    AXIS_COMBINED_VERTICAL_CALIBRATION : UINT := 25;
    AXIS_COMBINED_VERTICAL_SAMPLE : UINT :=26;
    AXIS_COMBINED_VERTICAL_VIRTUAL : UINT :=27;
    
    AXIS_HORIZONTAL_CALIBRATION : UINT :=28;
    AXIS_HORIZONTAL_SAMPLE : UINT :=29;
    AXIS_HORIZONTAL_VIRTUAL : UINT :=30;
    

END_VAR

// ---- tc_mca_std_lib/GVLs/GVL.TcGVL
VAR_GLOBAL
    // Semantic version in machine-readable format.
    // Update it and commit it immediatly before setting a tag
    nVersionMajor: UINT := 2; // Major Version
    nVersionMinor: UINT := 0; // Minor Version
    nVersionPatch: UINT := 2; // Patch level
    astAxes: ARRAY [1..GVL_APP.nAXIS_NUM] OF ST_AxisStruct; //Array of ST_AxisStruct for holding axis parameters and controls
    astPneumaticAxes: ARRAY [1..GVL_APP.nPNEUMATIC_AXIS_NUM] OF ST_PneumaticAxisStruct; //Array of ST_PneumaticAxisStruct for holding pneumatic axis parameters and controls
    iAxis: UINT; //Index for for loops while going through axes
    iPneumaticAxis: UINT := 1; //Index for for loops while going through pneumatic axes
    fbGetCurTaskIndex: GETCURTASKINDEX;
    bLocalMode: BOOL;
END_VAR

VAR_GLOBAL CONSTANT
    nMAX_AXIS_NAME: UINT := 32;
END_VAR

VAR_GLOBAL PERSISTENT
    astAxesPersistent: ARRAY [1..GVL_APP.nAXIS_NUM] OF ST_AxisPersistent;
END_VAR

// ---- POUs/MAIN.TcPOU
PROGRAM MAIN
VAR
    sVersion: STRING := '1.0.0';
    aIAxes: ARRAY [1..GVL_APP.nAXIS_NUM] OF I_Axis;
    afbAxes: ARRAY [1..GVL_APP.nAXIS_NUM] OF FB_Axis;
    afbPneumaticAxes: ARRAY [1..GVL_APP.nPNEUMATIC_AXIS_NUM] OF FB_PneumaticAxis;
    hmiAxisSelection: INT := 1; //Not possible to use local hmi variables for array indexes
    hmiPneumaticAxisSelection: INT := 1;
//Startup, Shutdown and UPS
    fbUPS: FB_S_UPS_CX51x0;
    eUpsMode: E_S_UPS_Mode := eSUPS_WrPersistData_Shutdown;
    eStartUp: (eColdStart, eReadAxisFeedbackType, eCheckReadDone, eExecuteRestore, eCheckRestore, eFinishRestore);
    bPositionRestoreDone: BOOL := FALSE;
    bRestoreExecute: BOOL := FALSE;
    bExecuteReadEncRefSys: BOOL := FALSE;
    nRetry: INT;
    iAxes: UINT; //index for for loops in Position recovery actions
    afbReadEncRefSys: ARRAY [1..GVL_APP.nAXIS_NUM] OF MC_ReadParameter;
    afbSetPosition: ARRAY [1..GVL_APP.nAXIS_NUM] OF MC_SetPosition;
    afbReadPositionBias: ARRAY [1..GVL_APP.nAXIS_NUM] OF MC_ReadParameter;
    afbWritePositionBias: ARRAY [1..GVL_APP.nAXIS_NUM] OF MC_WriteParameter;
    fbGetDeviceIdentification: FB_GetDeviceIdentificationEx;
    
    
    
END_VAR

VAR PERSISTENT
    bRestoreOnStartup: BOOL;
END_VAR

POSITION_RECOVERY();
PROG();
AXES();

ACTION AXES:
//First cycle, assign FB_axis to interface array
IF _TaskInfo[fbGetCurTaskIndex.index].FirstCycle THEN
    FOR GVL.iAxis := 1 TO GVL_APP.nAXIS_NUM DO
        afbAxes[GVL.iAxis].stAxis REF= astAxes[GVL.iAxis];
        aIAxes[GVL.iAxis] := afbAxes[GVL.iAxis];
    END_FOR
    //Custom axis types defined and linked to aiAxes here
      //FB_CustomAxis extends FB_axis
        //fbCustomAxis.stAxis REF= astAxes[x];
        //aIAxes[x] := fbCustomAxis;
END_IF

//Execute FB_Axis logic
FOR GVL.iAxis := 1 TO GVL_APP.nAXIS_NUM DO
    aIAxes[GVL.iAxis].Run();
END_FOR

//Execute Pneumatic Axis logic
FOR GVL.iPneumaticAxis := 1 TO GVL_APP.nPNEUMATIC_AXIS_NUM DO
    afbPneumaticAxes[GVL.iPneumaticAxis](stPneumaticAxisStruct := GVL.astPneumaticAxes[GVL.iPneumaticAxis]);
END_FOR
END_ACTION

ACTION CHECK_UPS:
fbUPS(eUpsMode := eUpsMode);

FOR iAxes := 1 TO GVL_APP.nAXIS_NUM DO
    //Read encoder position BIAS
    IF astAxes[iAxes].stStatus.bAxisInitialized THEN
        afbReadPositionBias[iAxes](Axis := GVL.astAxes[iAxes].Axis,
                        Enable := TRUE,
                        ReadMode:= READMODE_CYCLIC,
                        ParameterNumber := E_AxisParameters.AxisEncoderOffset);
    END_IF
END_FOR

IF eGlobalSUpsState = eSUPS_PowerFailure THEN
    //first cycle of powerfailure
    //execute code that should only be done once with each powerfailure, i.e. increase powerfailure counter
    bRestoreOnStartup := TRUE;
    STORE_PERSISTENT();
    RETURN;
ELSIF eGlobalSUpsState <> eSUPS_PowerOK THEN
    //next cycles of powerfailure
    //skip regular code execution for the remaining cycles of the powerfailure/writing of persistent data/quick shutdown...
    RETURN;
END_IF
END_ACTION

ACTION POSITION_RECOVERY:
fbGetDeviceIdentification(bExecute := TRUE);
IF (fbGetDeviceIdentification.stDevIdent.strHardwareSerialNo <> '') THEN
    CHECK_UPS();
    RESTORE_POSITIONS();
END_IF
END_ACTION

ACTION PROG:
//Get task index for Axes parameters initialization.
GVL.fbGetCurTaskIndex();

//Call the programs that are defined in the "Application Specific" folder.
//Create as many programs in that folder as axes and applications you have or need

//Axes initial parameters and program
//Axis_Template();
//Pneumatics_Template();

//Application program calls
//Application_Template();
PLC_SAFETY_LOGIC();

Horizontal_Translation();
Vertical_Translation_Y2();
Vertical_Translation_Y1();
Rotation();

Combined_Vertical();


Drad_External();
Drad_Internal();
Doff_Angled();
Doff_Parallel();
Dtank_Internal_Offset_Angle();
Dtank_Length();
Dtank_Pivot_To_Window();
Delta();
Tau();
Drad();
Measurement_Angle();
Rotation_Calibration();
Rotation_Sample();
Horizontal_Calibration();
Horizontal_Sample();
Combined_Vertical_Calibration();
Combined_Vertical_Sample();
Measurement_Angle_Offset();


Rotation_Virtual();
Combined_Vertical_Virtual();
Horizontal_Virtual();




INTER_LOGIC();
VirtualSpeedOverrides();
//Slit setup
Slit_North();
Slit_South();
Slit_East();
Slit_West();
Slit_3();

Inclinometer();
END_ACTION

ACTION RESTORE_POSITIONS:
//This ACT will restore the position of an incremental axis on startup with the act position it read before losing power.
//It checks the type of axis, 0=incremental, and that the axis was stationary at shut down.
//Because 0 equates to incremental we also need to check that the data is valid, otherwise by default it would restore all axes.
//By default an axis will not restore the position unless it is set to opt-in, i.e. GVL.aAxes[iAxes].stConfig.eRestorePosition is non-zero.
//This needs to be initialised somewhere in TwinCAT code otherwise it will not be available at start up.
//A restore will only be performed on a loss of power, this code shouldn't make any changes on a reset cold, a rest origin or a download.
//There is a enum to allow for different types of restore modes, currently only one is implemented.
//0 'DontRestore'
//1 'RestoreWithoutHome' -restores the position using a set position fb and does not set the home bit in the axis struct.
//Note from Beckhoff: "A maximum of 1 MB persistent data can be reliably saved over the entire service life."
//Encoder Reference system types: https://infosys.beckhoff.com/english.php?content=../content/1033/tf50x0_tc3_nc_ptp/3439907723.html&id=
//INCREMENTAL=0;
//ABSOLUTE=1;
//ABSOLUTE (modulo)=2;
//ABSOLUTE MULTITURN RANGE (with single overflow)=3;
//INCREMENTAL (singleturn absolute)=4;
//ABSOLUTE SINGLETURN RANGE (with single overflow)=5;


IF bRestoreOnStartup AND eGlobalSUpsState = eSUPS_PowerOK THEN
    bRestoreOnStartup := FALSE;
    bRestoreExecute := TRUE;
END_IF

//Upon startup bPositionRestoreDone will be set to FALSE, after successfully completing the following code it will be set TRUE
//and should stay TRUE for the rest of the time the PLC is operational, thus this routine should only be completed once.
IF bRestoreExecute AND NOT bPositionRestoreDone THEN
    //Cycle through function blocks that read the encoder reference system i.e. whether axis is incremental or absolute
    FOR iAxes := 1 TO GVL_APP.nAXIS_NUM DO
         afbReadEncRefSys[iAxes](
            Axis := GVL.astAxes[iAxes].Axis,
            ParameterNumber := MC_AxisParameter.AxisEncoderReferenceSystem,
            ReadMode := E_READMODE.READMODE_ONCE);
    END_FOR

    //Cycle through set position and MC_WritePArameter function blocks for each axis
    FOR iAxes := 1 TO GVL_APP.nAXIS_NUM DO
        afbSetPosition[iAxes](
            Axis := GVL.astAxes[iAxes].Axis,
            Position := astAxesPersistent[iAxes].fPositionAtShutdown);

        afbWritePositionBias[iAxes](
            Axis:= GVL.astAxes[iAxes].Axis,
            ParameterNumber:= E_AxisParameters.AxisEncoderOffset,
            Value:= astAxesPersistent[iAxes].fEncoderBiasAtShutdown);
    END_FOR

    CASE eStartUp OF
        eColdStart:
            //First cycle of the PLC, do nothing just give one cycle for variables to initialise
            IF NOT bPositionRestoreDone THEN
                eStartUp := eReadAxisFeedbackType;
                nRetry := 0;
            END_IF

        eReadAxisFeedbackType:
            //Exectute the function blocks to read the encoder reference system (0=inc OR 1=ABS)
            FOR iAxes := 1 TO GVL_APP.nAXIS_NUM DO
                afbReadEncRefSys[iAxes].Enable := TRUE;
                eStartUp := eCheckReadDone;
            END_FOR

        eCheckReadDone:
            //Check the encoder reference system has been read for all axis -> if busy then continue with PLC cycle and check again next time.
            //If afbReadEncRefSys not started then go back a step.
            //If any axes result in an error the code will get stuck here, this happens if GVL_APP.nAXIS_NUM is not set correctly
            FOR iAxes := 1 TO GVL_APP.nAXIS_NUM DO
                IF NOT afbReadEncRefSys[iAxes].Valid THEN
                    IF afbReadEncRefSys[iAxes].Busy THEN
                        //Exit MAIN.STARTUP Action and wait till next cycle, needs to cycle through whole program in order for data to update
                        RETURN;
                    ELSE
                        //Sometimes the code gets here and the afbReadEncRefSys[iAxes] misses the rising edge. If  the code gets here it means
                        //valid=FALSE and .busy=FALSE which indicateds the FB probably hasn't started and thus needs to see a rising edge.
                        //Set execute to low, Exit MAIN.STARTUP and go back a step in the CASE statement.
                        afbReadEncRefSys[iAxes].Enable := FALSE;
                        eStartUp := eReadAxisFeedbackType;
                        nRetry := nRetry + 1; //counter used for troubleshooting to see how many cycles it takes before afbReadEncRefSys function blocks are read correctly
                        RETURN;
                    END_IF
                END_IF
            END_FOR
            //If the code gets here all axes have .valid=TRUE for all axes
            eStartUp := eExecuteRestore;

        eExecuteRestore:
            //Execute position and encoder BIAS restore by setting Execute = TRUE
           FOR iAxes := 1 TO GVL_APP.nAXIS_NUM DO
                IF GVL.astAxes[iAxes].stConfig.eRestorePosition = E_RestorePosition.eRestoreWithoutHome THEN
                    //Restore position value for incremental encoders
                    IF NOT astAxesPersistent[iAxes].bMovingAtShutdown AND
                    (afbReadEncRefSys[iAxes].Value = 0 OR
                     afbReadEncRefSys[iAxes].Value = 2 OR
                     afbReadEncRefSys[iAxes].Value = 4) THEN
                       afbSetPosition[iAxes].Execute := TRUE;
                    //Restore encoder position BIAS for absolute encoders
                    ELSIF afbReadEncRefSys[iAxes].Value = 1 OR
                    afbReadEncRefSys[iAxes].Value = 3 OR
                    afbReadEncRefSys[iAxes].Value = 5 THEN
                       afbWritePositionBias[iAxes].Execute := TRUE;
                    END_IF
                ELSE
                    RETURN;
                END_IF
            END_FOR
            eStartUp := eCheckRestore;


        eCheckRestore:
            //Check the set position and write enocder BIAS fbs are finished
            //Nothing actually happens if the restore is not done, the code just returns from here each cycle and the
            //bPositionRestoreDone will never get set to TRUE and will take up cycle time
            FOR iAxes := 1 TO GVL_APP.nAXIS_NUM DO
                IF GVL.astAxes[iAxes].stConfig.eRestorePosition = E_RestorePosition.eRestoreWithoutHome THEN
                    IF NOT astAxesPersistent[iAxes].bMovingAtShutdown AND
                    (afbReadEncRefSys[iAxes].Value = 0 OR
                     afbReadEncRefSys[iAxes].Value = 2 OR
                     afbReadEncRefSys[iAxes].Value = 4) THEN
                        IF NOT afbSetPosition[iAxes].Done THEN
                            afbSetPosition[iAxes].Execute := FALSE;
                            eStartUp := eExecuteRestore;
                            RETURN;
                        END_IF
                     ELSIF afbReadEncRefSys[iAxes].Value = 1 OR
                     afbReadEncRefSys[iAxes].Value = 3 OR
                     afbReadEncRefSys[iAxes].Value = 5 THEN
                        IF NOT afbWritePositionBias[iAxes].Done THEN
                            afbWritePositionBias[iAxes].Execute := FALSE;
                            eStartUp := eExecuteRestore;
                            RETURN;
                        END_IF
                    END_IF
                ELSE
                    RETURN;
                END_IF
            END_FOR
            eStartUp :=  eFinishRestore;

        eFinishRestore:
            //Remove execute = TRUE for afbRestorePosition and fbWritePositionBias
            FOR iAxes := 1 TO GVL_APP.nAXIS_NUM DO
                afbSetPosition[iAxes].Execute := FALSE;
                afbWritePositionBias[iAxes].Execute := FALSE;
                bPositionRestoreDone := TRUE;
                bRestoreExecute := FALSE;
            END_FOR
    END_CASE
END_IF
END_ACTION

ACTION STORE_PERSISTENT:
FOR iAxes := 1 TO GVL_APP.nAXIS_NUM DO
    //Store Position beofre shutdown
    astAxesPersistent[iAxes].fPositionAtShutdown := GVL.astAxes[iAxes].Axis.NcToPlc.ActPos;

    //Store encoder position BIAS at shutdown
    astAxesPersistent[iAxes].fEncoderBiasAtShutdown := afbReadPositionBias[iAxes].Value;

    //Store value of moving at shutdown
    IF GVL.astAxes[iAxes].Axis.Status.StandStill OR GVL.astAxes[iAxes].Axis.Status.Disabled THEN
        astAxesPersistent[iAxes].bMovingAtShutdown := FALSE;
    ELSE
        astAxesPersistent[iAxes].bMovingAtShutdown := TRUE;
    END_IF
END_FOR
END_ACTION

END_PROGRAM

// ---- tc_mca_std_lib/POUs/Motion/FB_Axis.TcPOU
//Function block to run a virtual drive with Nc
FUNCTION_BLOCK FB_Axis IMPLEMENTS I_axis
VAR
    _stAxis: REFERENCE TO ST_AxisStruct; // Local property pointer for axis structure
    astMcStatus: ARRAY[1..nMCSTATUS_ARRAY_SIZE] OF POINTER TO ST_McStatus; //Array of all MC status signals defined in FB_init

    fbPower: MC_Power;
    stMcStatusPower: ST_McStatus;

    fbStop: MC_Stop;
    stMcStatusStop: ST_McStatus;

    fbHalt: MC_Halt;
    stMcStatusHalt: ST_McStatus;

    fbReset: MC_Reset;
    stMcStatusReset: ST_McStatus;

    fbMoveAbsolute: MC_MoveAbsolute;
    stMcStatusMoveAbsolute: ST_McStatus;

    fbMoveRelative: MC_MoveRelative;
    stMcStatusMoveRelative: ST_McStatus;

    fbMoveVelocity: MC_MoveVelocity;
    stMcStatusMoveVelocity: ST_McStatus;

    fbMoveModulo: MC_MoveModulo;
    stMcStatusMoveModulo: ST_McStatus;

    fbHome: FB_Homing;
    stMcStatusHome: ST_McStatus;

    fbReadParameter: MC_ReadParameter;
    stMcStatusReadParameter: ST_McStatus;

    fbWriteParameter: MC_WriteParameter;
    stMcStatusWriteParameter: ST_McStatus;

    fbGearIn: MC_GearIn;
    stMcStatusGearIn: ST_McStatus;

    fbGearOut: MC_GearOut;
    stMcStatusGearOut: ST_McStatus;

    stMasterAxis: ST_GearAxis := (nIndex := 1, fRatio := 0);
    nSlaveAxesIndex: UINT;
    nAxisIndex: UINT;
    nMultiMastersAxesIndex: UINT;

    fbGearInMultiMaster: MC_GearInMultiMaster;
    stMcStatusGearInMultiMaster: ST_McStatus;

    //Variables for holding limits during homing
    bWaitForStopAfterLimitHit: BOOL := FALSE;
    fbRemovePowerTimer: TOF;

    //Dedicated NC parameter read FBs
    fbReadAxisVeloManSlow: MC_ReadParameter;
    fbReadAxisVeloManFast: MC_ReadParameter;
    fbReadHomingVelToCam: MC_ReadParameter;
    fbReadHomingVelFromCam: MC_ReadParameter;
    fbReadAxisVeloMax: MC_ReadParameter;
    fbReadAxisMaxAcc: MC_ReadParameter;
    fbReadAxisMaxDec: MC_ReadParameter;
    fbReadAxisAcc: MC_ReadParameter;
    fbReadAxisDec: MC_ReadParameter;
    fbReadEnMinSoftPosLimit: MC_ReadParameter;
    fbReadEnMaxSoftPosLimit: MC_ReadParameter;
    fbReadMinSoftPosLimit: MC_ReadParameter;
    fbReadMaxSoftPosLimit: MC_ReadParameter;
    fbReadEnPositionLagMonitoring: MC_ReadParameter;
    fbReadAxisMaxPosLagValue: MC_ReadParameter;
    fbReadEnTargetPositionMonitoring: MC_ReadParameter;
    fbReadTargetPositionWindow: MC_ReadParameter;

    //Edge detection triggers for statuses
    fbDoneRTrig: R_TRIG;
    fbErrorRTrig: R_TRIG;
    fbCommandAbortedRTrig: R_TRIG;
    fbInVelocityRTrig: R_TRIG;
    fbInVelocityFTrig: F_TRIG;
    fbExecuteRTrig: R_TRIG;
    fbStopFinishedRiseEdge: R_TRIG;
    fbHaltFinishedRiseEdge: R_TRIG;
    fbResetFinishedRiseEdge: R_TRIG;

END_VAR
VAR CONSTANT
    nRATIO_DENOMINATOR_DEFAULT: UINT := 1;
    nNO_GEARING: UINT := 0;
    nMCSTATUS_ARRAY_SIZE: UINT := 13;
    nMULTI_MASTER_MAX_AXES: UINT := 4;
END_VAR

METHOD EndOfCycle : BOOL

_stAxis.stControl.bExecute := FALSE;
END_METHOD

METHOD FB_init : BOOL
VAR_INPUT
    bInitRetains: BOOL; // if TRUE, the retain variables are initialized (warm start / cold start)
    bInCopyCode: BOOL; // if TRUE, the instance afterwards gets moved into the copy code (online change)
END_VAR

//Copy address locations for statuses to an array to allow for easier checking of statuses
astMcStatus[1] := ADR(stMcStatusPower);
astMcStatus[2] := ADR(stMcStatusStop);
astMcStatus[3] := ADR(stMcStatusHalt);
astMcStatus[4] := ADR(stMcStatusReset);
astMcStatus[5] := ADR(stMcStatusMoveAbsolute);
astMcStatus[6] := ADR(stMcStatusMoveRelative);
astMcStatus[7] := ADR(stMcStatusMoveVelocity);
astMcStatus[8] := ADR(stMcStatusMoveModulo);
astMcStatus[9] := ADR(stMcStatusHome);
astMcStatus[10] := ADR(stMcStatusGearInMultiMaster);
astMcStatus[11] := ADR(stMcStatusGearOut);
astMcStatus[12] := ADR(stMcStatusReadParameter);
astMcStatus[13] := ADR(stMcStatusWriteParameter);
END_METHOD

METHOD mControl_GearInMultiMaster : ST_McStatus

fbGearInMultiMaster.Options.AdvancedSlaveDynamics := TRUE;
fbGearInMultiMaster.Options.SyncMode := E_GearInMultiMasterSyncMode.POSSYNC2;
IF _stAxis.stControl.eCommand = E_MotionFunctions.eGearInMultiMaster THEN
    fbGearInMultiMaster.Enable := _stAxis.stControl.bExecute;
END_IF

IF _stAxis.stControl.eCommand = E_MotionFunctions.eGearInMultiMaster AND _stAxis.stControl.bExecute AND NOT _stAxis.Axis.Status.Coupled THEN
    //Latch master references
    FOR nMultiMastersAxesIndex := 1 TO nMULTI_MASTER_MAX_AXES DO
        IF _stAxis.stConfig.astMultiMasterAxis[nMultiMastersAxesIndex].nIndex > 0 AND _stAxis.stConfig.astMultiMasterAxis[nMultiMastersAxesIndex].nIndex <= GVL_APP.nAXIS_NUM THEN
            _stAxis.stConfig.astMultiMasterAxisLatched[nMultiMastersAxesIndex].nIndex := _stAxis.stConfig.astMultiMasterAxis[nMultiMastersAxesIndex].nIndex;
        END_IF
    END_FOR
    //Latch gear ratios
    FOR nMultiMastersAxesIndex := 1 TO nMULTI_MASTER_MAX_AXES DO
        _stAxis.stConfig.astMultiMasterAxisLatched[nMultiMastersAxesIndex].fRatio := _stAxis.stConfig.astMultiMasterAxis[nMultiMastersAxesIndex].fRatio;
    END_FOR
    //Transfer gear ratios to FB
    fbGearInMultiMaster.GearRatio1 := _stAxis.stConfig.astMultiMasterAxisLatched[1].fRatio;
    fbGearInMultiMaster.GearRatio2 := _stAxis.stConfig.astMultiMasterAxisLatched[2].fRatio;
    fbGearInMultiMaster.GearRatio3 := _stAxis.stConfig.astMultiMasterAxisLatched[3].fRatio;
    fbGearInMultiMaster.GearRatio4 := _stAxis.stConfig.astMultiMasterAxisLatched[4].fRatio;
    fbGearInMultiMaster.Enable := TRUE;
END_IF

fbGearInMultiMaster(Slave := _stAxis.Axis,
    Master1 := GVL.astAxes[_stAxis.stConfig.astMultiMasterAxisLatched[1].nIndex].Axis,
    Master2 := GVL.astAxes[_stAxis.stConfig.astMultiMasterAxisLatched[2].nIndex].Axis,
    Master3 := GVL.astAxes[_stAxis.stConfig.astMultiMasterAxisLatched[3].nIndex].Axis,
    Master4 := GVL.astAxes[_stAxis.stConfig.astMultiMasterAxisLatched[4].nIndex].Axis);
fbGearInMultiMaster.Enable:= FALSE;

IF fbGearInMultiMaster.InGear THEN
    mStatus_MultiGearing();
END_IF

IF fbGearInMultiMaster.Error THEN
    fbGearInMultiMaster.Enable := FALSE;
END_IF

mControl_GearInMultiMaster.Active := fbGearInMultiMaster.Active;
mControl_GearInMultiMaster.Done := fbGearInMultiMaster.InGear;
mControl_GearInMultiMaster.Busy := fbGearInMultiMaster.Busy;
mControl_GearInMultiMaster.Error := fbGearInMultiMaster.Error;
mControl_GearInMultiMaster.ErrorID := fbGearInMultiMaster.ErrorID;
mControl_GearInMultiMaster.CommandAborted := fbGearInMultiMaster.CommandAborted;

IF fbGearInMultiMaster.Error THEN
    _stAxis.stError.nGearInMultiMasterErrorID := fbGearInMultiMaster.ErrorID; //Set the error
END_IF
END_METHOD

METHOD mControl_GearOut : ST_McStatus

IF _stAxis.stControl.eCommand = E_MotionFunctions.eGearOut THEN
    fbGearOut.Execute := _stAxis.stControl.bExecute;
END_IF

fbGearOut(Slave := _stAxis.Axis);
fbGearOut.Execute := FALSE;

//Clear ratios from single and multi master gearing
IF fbGearOut.Done THEN
    //Clear slave ratio from master axis slave array
    mStatus_MultiGearing();
    FOR nSlaveAxesIndex := 1 TO GVL_APP.nAXIS_NUM DO
        GVL.astAxes[nSlaveAxesIndex].stConfig.afMultiSlaveAxisRatio[GVL.iAxis] := nNO_GEARING;
    END_FOR
END_IF

mControl_GearOut.Done := fbGearOut.Done;
mControl_GearOut.Busy := fbGearOut.Busy;
mControl_GearOut.Error := fbGearOut.Error;
mControl_GearOut.ErrorID := fbGearOut.ErrorID;

IF fbGearOut.Error THEN
    _stAxis.stError.nGearOutErrorID := fbGearOut.ErrorID; //Set the error
END_IF
END_METHOD

METHOD mControl_Home : ST_McStatus

IF _stAxis.stControl.eCommand = E_MotionFunctions.eHome THEN
    fbHome.bExecute := _stAxis.stControl.bExecute;
END_IF


fbHome.eHomeSeq := _stAxis.stConfig.eHomeSeq;
fbHome.fHomePosition := _stAxis.stConfig.fHomePosition;
fbHome.fHomeFinishDistance := _stAxis.stConfig.fHomeFinishDistance;
fbHome(
    Axis := _stAxis.Axis,
    bLimitBwd := _stAxis.stInputs.bLimitBwd,
    bLimitFwd := _stAxis.stInputs.bLimitFwd,
    bHomeSensor := _stAxis.stInputs.bHomeSensor,
    stConfig := _stAxis.stConfig);
fbHome.bExecute := FALSE;

mControl_Home.Busy := fbHome.bBusy;
mControl_Home.CommandAborted := fbHome.bCommandAborted;
mControl_Home.Done := fbHome.bDone;
mControl_Home.Error := fbHome.bError;
mControl_Home.ErrorID := fbHome.nErrorId;

IF fbHome.bError THEN
    _stAxis.stError.nHomeErrorID := fbHome.nErrorID; //Set the error
END_IF
END_METHOD

METHOD mControl_LimitHitTimer : BOOL

//Timer for keeping power on after limit switch hit, needed for homing routines - if power is lost routines are aborted
fbRemovePowerTimer(IN := _stAxis.stInputs.bLimitFwd AND _stAxis.stInputs.bLimitBwd, PT := T#100MS);

IF stMcStatusHome.Busy AND (fbRemovePowerTimer.Q OR _stAxis.Axis.NcToPlc.AxisState = 5) THEN //5=PHASE_ACCNEG
    bWaitForStopAfterLimitHit := TRUE;
ELSE
    bWaitForStopAfterLimitHit := FALSE;
END_IF
END_METHOD

METHOD mControl_LimitLinking : BOOL

_stAxis.stStatus.bFwEnabled := _stAxis.stInputs.bLimitFwd; //Moved to linking code. Should not say enabled if not enabled
_stAxis.stStatus.bBwEnabled := _stAxis.stInputs.bLimitBwd;
_stAxis.stStatus.bInterlockedFwd := _stAxis.stControl.bInterlockFwd;
_stAxis.stStatus.bInterlockedBwd := _stAxis.stControl.bInterlockBwd;

//Multimaster limit linking
FOR nAxisIndex := 1 TO GVL_APP.nAXIS_NUM DO
    IF (_stAxis.stConfig.afMultiSlaveAxisRatio[nAxisIndex] <> 0) THEN
        _stAxis.stStatus.bFwEnabled := _stAxis.stStatus.bFwEnabled AND SEL(_stAxis.stConfig.afMultiSlaveAxisRatio[nAxisIndex] > 0, GVL.astAxes[nAxisIndex].stStatus.bBwEnabled, GVL.astAxes[nAxisIndex].stStatus.bFwEnabled);
        _stAxis.stStatus.bBwEnabled := _stAxis.stStatus.bBwEnabled AND SEL(_stAxis.stConfig.afMultiSlaveAxisRatio[nAxisIndex] > 0, GVL.astAxes[nAxisIndex].stStatus.bFwEnabled, GVL.astAxes[nAxisIndex].stStatus.bBwEnabled);
    END_IF
END_FOR
END_METHOD

METHOD mControl_Power : ST_McStatus

fbPower.Enable := _stAxis.stControl.bEnable;
fbPower.Enable_Negative := (_stAxis.stStatus.bBwEnabled OR bWaitForStopAfterLimitHit) AND NOT _stAxis.stStatus.bInterlockedBwd;
fbPower.Enable_Positive := (_stAxis.stStatus.bFwEnabled OR bWaitForStopAfterLimitHit) AND NOT _stAxis.stStatus.bInterlockedFwd;
fbPower.Override := _stAxis.stConfig.fOverride;

fbPower(Axis := _stAxis.Axis);

mControl_Power.Error := fbPower.Error;

IF fbPower.Error THEN
    _stAxis.stError.nPowerErrorID := fbPower.ErrorID; //Set the error
END_IF
END_METHOD

METHOD mControl_Reset : ST_McStatus
VAR
    i: UINT;
END_VAR
fbReset.Execute := _stAxis.stControl.bReset;

fbReset(Axis := _stAxis.Axis);
IF fbReset.Done THEN
    _stAxis.stStatus.bError := FALSE;
    FOR i := 1 TO nMCSTATUS_ARRAY_SIZE DO
        //If there's an error present propagate
        _stAxis.stStatus.nErrorID := 0;
    END_FOR
END_IF

mControl_Reset.Busy := fbReset.Busy;
mControl_Reset.Done := fbReset.Done;
mControl_Reset.Error := fbReset.Error;
mControl_Reset.ErrorID := fbReset.ErrorID;

IF fbReset.Error THEN
    _stAxis.stError.nResetErrorID := fbReset.ErrorID; //Set the error
END_IF

fbResetFinishedRiseEdge(CLK:=fbReset.Done OR fbReset.Error);
IF fbResetFinishedRiseEdge.Q OR fbReset.Done THEN
    _stAxis.stControl.bReset := FALSE;
END_IF
END_METHOD

METHOD mMove_Halt : ST_McStatus

fbHalt.Deceleration := _stAxis.stControl.fDeceleration;
fbHalt.Execute := _stAxis.stControl.bHalt;

fbHalt(Axis := _stAxis.Axis);

mMove_Halt.Busy := fbHalt.Busy;
mMove_Halt.Done := fbHalt.Done;
mMove_Halt.Error := fbHalt.Error;
mMove_Halt.ErrorID := fbHalt.ErrorID;
mMove_Halt.Active := fbHalt.Active;
mMove_Halt.CommandAborted := fbHalt.CommandAborted;

IF fbHalt.Error THEN
    _stAxis.stError.nHaltErrorID := fbHalt.ErrorID; //Set the error
END_IF

//Execution of fbHalt ended
fbHaltFinishedRiseEdge(CLK:=fbHalt.Done OR fbHalt.Error OR fbHalt.CommandAborted);
IF fbHaltFinishedRiseEdge.Q OR fbHalt.Done OR fbHalt.CommandAborted THEN
    _stAxis.stControl.bHalt := FALSE;
END_IF
END_METHOD

METHOD mMove_MoveAbsolute : ST_McStatus

IF _stAxis.stControl.eCommand = E_MotionFunctions.eMoveAbsolute THEN
    fbMoveAbsolute.Execute := _stAxis.stControl.bExecute;
END_IF

fbMoveAbsolute.Position := _stAxis.stControl.fPosition;
fbMoveAbsolute.Velocity := ABS(_stAxis.stControl.fVelocity);
fbMoveAbsolute.Acceleration := _stAxis.stControl.fAcceleration;
fbMoveAbsolute.Deceleration := _stAxis.stControl.fDeceleration;

fbMoveAbsolute(Axis := _stAxis.Axis);
fbMoveAbsolute.Execute := FALSE;

mMove_MoveAbsolute.Active := fbMoveAbsolute.Active;
mMove_MoveAbsolute.Done := fbMoveAbsolute.Done;
mMove_MoveAbsolute.Busy := fbMoveAbsolute.Busy;
mMove_MoveAbsolute.Error := fbMoveAbsolute.Error;
mMove_MoveAbsolute.ErrorID := fbMoveAbsolute.ErrorID;
mMove_MoveAbsolute.CommandAborted := fbMoveAbsolute.CommandAborted;

IF fbMoveAbsolute.Error THEN
    _stAxis.stError.nMoveAbsoluteErrorID := fbMoveAbsolute.ErrorID; //Set the error
END_IF
END_METHOD

METHOD mMove_MoveModulo : ST_McStatus

IF _stAxis.stControl.eCommand = E_MotionFunctions.eMoveModulo THEN
    fbMoveModulo.Execute := _stAxis.stControl.bExecute;
END_IF

fbMoveModulo.Position := _stAxis.stControl.fPosition;
fbMoveModulo.Velocity := ABS(_stAxis.stControl.fVelocity);
fbMoveModulo.Acceleration := _stAxis.stControl.fAcceleration;
fbMoveModulo.Deceleration := _stAxis.stControl.fDeceleration;

fbMoveModulo(Axis := _stAxis.Axis);
fbMoveModulo.Execute := FALSE;

mMove_MoveModulo.Active := fbMoveModulo.Active;
mMove_MoveModulo.Done := fbMoveModulo.Done;
mMove_MoveModulo.Busy := fbMoveModulo.Busy;
mMove_MoveModulo.Error := fbMoveModulo.Error;
mMove_MoveModulo.ErrorID := fbMoveModulo.ErrorID;
mMove_MoveModulo.CommandAborted := fbMoveModulo.CommandAborted;

IF fbMoveModulo.Error THEN
    _stAxis.stError.nMoveModuloErrorID := fbMoveModulo.ErrorID; //Set the error
END_IF
END_METHOD

METHOD mMove_MoveRelative : ST_McStatus

IF _stAxis.stControl.eCommand = E_MotionFunctions.eMoveRelative THEN
    fbMoveRelative.Execute := _stAxis.stControl.bExecute;
END_IF

fbMoveRelative.Distance := _stAxis.stControl.fPosition;
fbMoveRelative.Velocity := ABS(_stAxis.stControl.fVelocity);
fbMoveRelative.Acceleration := _stAxis.stControl.fAcceleration;
fbMoveRelative.Deceleration := _stAxis.stControl.fDeceleration;

fbMoveRelative(Axis := _stAxis.Axis);
fbMoveRelative.Execute := FALSE;

mMove_MoveRelative.Active := fbMoveRelative.Active;
mMove_MoveRelative.Done := fbMoveRelative.Done;
mMove_MoveRelative.Busy := fbMoveRelative.Busy;
mMove_MoveRelative.Error := fbMoveRelative.Error;
mMove_MoveRelative.ErrorID := fbMoveRelative.ErrorID;
mMove_MoveRelative.CommandAborted := fbMoveRelative.CommandAborted;

IF fbMoveRelative.Error THEN
    _stAxis.stError.nMoveRelativeErrorID := fbMoveRelative.ErrorID; //Set the error
END_IF
END_METHOD

METHOD mMove_MoveVelocity : ST_McStatus

IF _stAxis.stControl.eCommand = E_MotionFunctions.eMoveVelocity THEN
    fbMoveVelocity.Execute := _stAxis.stControl.bExecute;
END_IF

fbMoveVelocity.Direction := SEL(_stAxis.stControl.fVelocity < 0, MC_Positive_Direction, MC_Negative_Direction);
fbMoveVelocity.Velocity := ABS(_stAxis.stControl.fVelocity);
fbMoveVelocity.Acceleration := _stAxis.stControl.fAcceleration;
fbMoveVelocity.Deceleration := _stAxis.stControl.fDeceleration;

fbMoveVelocity(Axis := _stAxis.Axis);
fbMoveVelocity.Execute:= FALSE;

mMove_MoveVelocity.Active := fbMoveVelocity.Active;
mMove_MoveVelocity.InVelocity := fbMoveVelocity.InVelocity;
mMove_MoveVelocity.Busy := fbMoveVelocity.Busy;
mMove_MoveVelocity.Error := fbMoveVelocity.Error;
mMove_MoveVelocity.ErrorID := fbMoveVelocity.ErrorID;
mMove_MoveVelocity.CommandAborted := fbMoveVelocity.CommandAborted;

IF fbMoveVelocity.Error THEN
    _stAxis.stError.nMoveVelocityErrorID := fbMoveVelocity.ErrorID; //Set the error
END_IF
END_METHOD

METHOD mMove_Stop : ST_McStatus

fbStop.Deceleration := _stAxis.stControl.fDeceleration;
fbStop.Execute := _stAxis.stControl.bStop;

fbStop(Axis := _stAxis.Axis);

mMove_Stop.Busy := fbStop.Busy;
mMove_Stop.Done := fbStop.Done;
mMove_Stop.Error := fbStop.Error;
mMove_Stop.ErrorID := fbStop.ErrorID;
mMove_Stop.Active := fbStop.Active;
mMove_Stop.CommandAborted := fbStop.CommandAborted;

IF fbStop.Error THEN
    _stAxis.stError.nStopErrorID := fbStop.ErrorID; //Set the error
END_IF

//Execution of fbStop ended
fbStopFinishedRiseEdge(CLK:=fbStop.Done OR fbStop.Error OR fbStop.CommandAborted);
IF fbStopFinishedRiseEdge.Q THEN
    _stAxis.stControl.bStop := FALSE;
END_IF
END_METHOD

METHOD mParameters_Init : BOOL

IF _stAxis.stConfig.bReadMcParametersValid AND NOT _stAxis.stStatus.bAxisInitialized THEN
    _stAxis.stControl.fAcceleration := _stAxis.stConfig.fDefaultAcc;
    _stAxis.stControl.fDeceleration := _stAxis.stConfig.fDefaultDec;
    _stAxis.stControl.fVelocity := _stAxis.stConfig.fVelocityDefaultFast;
    _stAxis.stControl.fJogVelocity := _stAxis.stConfig.fVelocityDefaultSlow;

    _stAxis.stStatus.bAxisInitialized := TRUE;
END_IF
END_METHOD

METHOD mParameters_ReadNc : BOOL

(*This act reads the MC parameters using an MC_ReadParameter FB FOR each variable
Intended TO be executed once every PLC cycle
Another FB is used TO trasnfer default axis parameters TO the stAxisStruct so
bReadValid is used TO halt that trasnfer UNTIL the parameters have been
read successfully. It may take a couple OF cycles once the PLC starts up.*)

//Slow jogging Velocity
fbReadAxisVeloManSlow(Axis := _stAxis.Axis,
                        Enable := TRUE,
                        ReadMode := READMODE_CYCLIC,
                        ParameterNumber := E_AxisParameters.AxisManualVelocitySlow,
                        Value => _stAxis.stConfig.fVelocityDefaultSlow);
//Fast jogging velocity
fbReadAxisVeloManFast(Axis := _stAxis.Axis,
                        Enable := TRUE,
                        ReadMode := READMODE_CYCLIC,
                        ParameterNumber := E_AxisParameters.AxisManualVelocityFast,
                        Value => _stAxis.stConfig.fVelocityDefaultFast);
//Homing velocity to Cam
fbReadHomingVelToCam(Axis := _stAxis.Axis,
                        Enable := TRUE,
                        ReadMode := READMODE_CYCLIC,
                        ParameterNumber := E_AxisParameters.AxisVelocityToCam,
                        Value => _stAxis.stConfig.fHomingVelToCam);
//Homing velocity from Cam
fbReadHomingVelFromCam(Axis := _stAxis.Axis,
                        Enable := TRUE,
                        ReadMode := READMODE_CYCLIC,
                        ParameterNumber := E_AxisParameters.AxisVelocityFromCam,
                        Value => _stAxis.stConfig.fHomingVelFromCam);
//Max velocity
fbReadAxisVeloMax(Axis := _stAxis.Axis,
                        Enable := TRUE,
                        ReadMode := READMODE_CYCLIC,
                        ParameterNumber := E_AxisParameters.AxisMaxVelocity,
                        Value => _stAxis.stConfig.fVeloMax);
//Max acceleration
fbReadAxisMaxAcc(Axis := _stAxis.Axis,
                        Enable := TRUE,
                        ReadMode := READMODE_CYCLIC,
                        ParameterNumber := E_AxisParameters.AxisMaximumAcceleration,
                        Value => _stAxis.stConfig.fMaxAcc);
//Max deceleration
fbReadAxisMaxDec(Axis := _stAxis.Axis,
                        Enable := TRUE,
                        ReadMode := READMODE_CYCLIC,
                        ParameterNumber := E_AxisParameters.AxisMaximumDeceleration,
                        Value => _stAxis.stConfig.fMaxDec);
//Default acceleration
fbReadAxisAcc(Axis := _stAxis.Axis,
                        Enable := TRUE,
                        ReadMode := READMODE_CYCLIC,
                        ParameterNumber := E_AxisParameters.AxisDefaultAcceleration,
                        Value => _stAxis.stConfig.fDefaultAcc);
//Default deceleration
fbReadAxisDec(Axis := _stAxis.Axis,
                        Enable := TRUE,
                        ReadMode := READMODE_CYCLIC,
                        ParameterNumber := E_AxisParameters.AxisDefaultDeceleration,
                        Value => _stAxis.stConfig.fDefaultDec);

//Soft limits enabled
fbReadEnMinSoftPosLimit(Axis := _stAxis.Axis,
                        Enable := TRUE,
                        ReadMode := READMODE_CYCLIC,
                        ParameterNumber := E_AxisParameters.EnableLimitBackward);
_stAxis.stConfig.bEnMinSoftPosLimit := LREAL_TO_BOOL(fbReadEnMinSoftPosLimit.Value);

fbReadEnMaxSoftPosLimit(Axis := _stAxis.Axis,
                        Enable := TRUE,
                        ReadMode := READMODE_CYCLIC,
                        ParameterNumber := E_AxisParameters.EnableLimitForward);
_stAxis.stConfig.bEnMaxSoftPosLimit := LREAL_TO_BOOL(fbReadEnMaxSoftPosLimit.Value);

//Soft limit values
fbReadMinSoftPosLimit(Axis := _stAxis.Axis,
                        Enable := TRUE,
                        ReadMode := READMODE_CYCLIC,
                        ParameterNumber := E_AxisParameters.SWLimitBackward,
                        Value => _stAxis.stConfig.fMinSoftPosLimit);
fbReadMaxSoftPosLimit(Axis := _stAxis.Axis,
                        Enable := TRUE,
                        ReadMode := READMODE_CYCLIC,
                        ParameterNumber := E_AxisParameters.SWLimitForward,
                        Value => _stAxis.stConfig.fMaxSoftPosLimit);

//Position Lag Monitoring
fbReadEnPositionLagMonitoring(Axis := _stAxis.Axis,
                        Enable := TRUE,
                        ReadMode := READMODE_CYCLIC,
                        ParameterNumber := E_AxisParameters.EnablePositionLagMonitoring);
_stAxis.stConfig.bEnPositionLagMonitoring := LREAL_TO_BOOL(fbReadEnPositionLagMonitoring.Value);

fbReadAxisMaxPosLagValue(Axis := _stAxis.Axis,
                        Enable := TRUE,
                        ReadMode := READMODE_CYCLIC,
                        ParameterNumber := E_AxisParameters.MaxPositionLag,
                        Value => _stAxis.stConfig.fMaxPosLagValue);

// Target Position Monitoring
fbReadEnTargetPositionMonitoring(Axis := _stAxis.Axis,
                        Enable := TRUE,
                        ReadMode := READMODE_CYCLIC,
                        ParameterNumber := E_AxisParameters.SWLimitBackward);
_stAxis.stConfig.bEnTargetPositionMonitoring := LREAL_TO_BOOL(fbReadEnTargetPositionMonitoring.Value);

fbReadTargetPositionWindow(Axis := _stAxis.Axis,
                        Enable := TRUE,
                        ReadMode := READMODE_CYCLIC,
                        ParameterNumber := E_AxisParameters.AxisTargetPositionWindow,
                        Value => _stAxis.stConfig.fTargetPositionWindow);

//All variables are valid
_stAxis.stConfig.bReadMcParametersValid := FALSE;
_stAxis.stConfig.bReadMcParametersValid := fbReadAxisVeloManSlow.Valid AND
    fbReadAxisVeloManFast.Valid AND
    fbReadHomingVelToCam.Valid AND
    fbReadHomingVelFromCam.Valid AND
    fbReadAxisVeloMax.Valid AND
    fbReadAxisAcc.Valid AND
    fbReadAxisDec.Valid AND
    fbReadEnMinSoftPosLimit.Valid AND
    fbReadEnMaxSoftPosLimit.Valid AND
    fbReadMinSoftPosLimit.Valid AND
    fbReadMaxSoftPosLimit.Valid AND
    fbReadEnPositionLagMonitoring.Valid AND
    fbReadAxisMaxPosLagValue.Valid AND
    fbReadEnTargetPositionMonitoring.Valid AND
    fbReadTargetPositionWindow.Valid;

//One of the variables has a read error
_stAxis.stConfig.bReadMcParametersError := fbReadAxisVeloManSlow.Error OR
    fbReadAxisVeloManFast.Error OR
    fbReadHomingVelToCam.Error OR
    fbReadHomingVelFromCam.Error OR
    fbReadAxisVeloMax.Error OR
    fbReadAxisAcc.Error OR
    fbReadAxisDec.Error OR
    fbReadEnMinSoftPosLimit.Error OR
    fbReadEnMaxSoftPosLimit.Error OR
    fbReadMinSoftPosLimit.Error OR
    fbReadMaxSoftPosLimit.Error OR
    fbReadEnPositionLagMonitoring.Error OR
    fbReadAxisMaxPosLagValue.Error OR
    fbReadEnTargetPositionMonitoring.Error OR
    fbReadTargetPositionWindow.Error;
END_METHOD

METHOD mParameters_ReadParameter : ST_McStatus

IF _stAxis.stControl.eCommand = E_MotionFunctions.eReadParameter THEN
    fbReadParameter.Enable := _stAxis.stControl.bExecute;
END_IF

fbReadParameter.ReadMode := E_READMODE.READMODE_ONCE;
fbReadParameter.ParameterNumber := _stAxis.stConfig.eAxisParameters;

fbReadParameter(Axis := _stAxis.Axis);
fbReadParameter.Enable := FALSE;

_stAxis.stconfig.fReadAxisParameter := fbReadParameter.Value;
mParameters_ReadParameter.Busy := fbReadParameter.Busy;
mParameters_ReadParameter.Done := fbReadParameter.Valid;
mParameters_ReadParameter.Error := fbReadParameter.Error;
mParameters_ReadParameter.ErrorID := fbReadParameter.ErrorID;

IF fbReadParameter.Error THEN
    _stAxis.stError.fbReadParameterErrorId := fbReadParameter.ErrorID;
END_IF
END_METHOD

METHOD mParameters_WriteParameter : ST_McStatus

IF _stAxis.stControl.eCommand = E_MotionFunctions.eWriteParameter THEN
    fbWriteParameter.Execute := _stAxis.stControl.bExecute;
END_IF

fbWriteParameter.ParameterNumber := _stAxis.stConfig.eAxisParameters;
fbWriteParameter.Value := _stAxis.stConfig.fWriteAxisParameter;

fbWriteParameter(Axis := _stAxis.Axis);
fbWriteParameter.Execute := FALSE;

mParameters_WriteParameter.Busy := fbWriteParameter.Busy;
mParameters_WriteParameter.Done := fbWriteParameter.Done;
mParameters_WriteParameter.Error := fbWriteParameter.Error;
mParameters_WriteParameter.ErrorID := fbWriteParameter.ErrorID;

IF fbWriteParameter.Error THEN
    _stAxis.stError.fbWriteParameterErrorId := fbWriteParameter.ErrorID;
END_IF
END_METHOD

METHOD mStatus_AxisStatus : BOOL

_stAxis.Axis.ReadStatus();
IF _stAxis.Axis.Status.OpMode.Modulo THEN
    _stAxis.stStatus.fActPosition := _stAxis.Axis.NcToPlc.ModuloActPos;
ELSE
    _stAxis.stStatus.fActPosition := _stAxis.Axis.NcToPlc.ActPos;
END_IF

_stAxis.stStatus.bGeared := _stAxis.Axis.Status.Coupled;
_stAxis.stStatus.bHomed := _stAxis.Axis.Status.Homed;
_stAxis.stStatus.bMoving := _stAxis.Axis.Status.Moving;
_stAxis.stStatus.fActVelocity := _stAxis.Axis.NcToPlc.ActVelo;
_stAxis.stStatus.bMovingForward := _stAxis.Axis.Status.PositiveDirection;
_stAxis.stStatus.bMovingBackward := _stAxis.Axis.Status.NegativeDirection;
_stAxis.stStatus.bInTargetPosition := _stAxis.Axis.Status.InTargetPosition;
_stAxis.stStatus.bEnabled := NOT(_stAxis.Axis.Status.Disabled);
END_METHOD

METHOD mStatus_Busy : BOOL
VAR
    i: UINT;
    tmpBusy: BOOL;
END_VAR

FOR i := 5 TO nMCSTATUS_ARRAY_SIZE DO
    tmpBusy := astMcStatus[i]^.Busy OR tmpBusy;
END_FOR
mStatus_Busy := tmpBusy;
END_METHOD

METHOD mStatus_CommandAborted : BOOL
VAR
    i: UINT;
    tmpCmdAborted: BOOL;
END_VAR

FOR i := 5 TO nMCSTATUS_ARRAY_SIZE DO
    tmpCmdAborted := astMcStatus[i]^.CommandAborted OR tmpCmdAborted;
END_FOR

fbCommandAbortedRTrig(CLK := tmpCmdAborted);
IF fbCommandAbortedRTrig.Q THEN
    _stAxis.stStatus.bCommandAborted := TRUE;
END_IF
END_METHOD

METHOD mStatus_Done : BOOL
VAR
    i: UINT;
    tmpDone: BOOL;
END_VAR

FOR i := 5 TO nMCSTATUS_ARRAY_SIZE DO
    tmpDone := astMcStatus[i]^.Done OR tmpDone;
END_FOR
//fbDoneRTrig(CLK:= mStatus_Done());
fbDoneRTrig(CLK := tmpDone);
IF fbDoneRTrig.Q THEN
    _stAxis.stStatus.bDone := TRUE;
END_IF
END_METHOD

METHOD mStatus_Error : BOOL
VAR
    i: UINT;
    tmpError: BOOL;
END_VAR

FOR i := 1 TO nMCSTATUS_ARRAY_SIZE DO
    tmpError := astMcStatus[i]^.Error OR tmpError;
END_FOR

fbErrorRTrig(CLK := tmpError);

IF _stAxis.Axis.Status.ErrorStop THEN
    _stAxis.stStatus.bError := _stAxis.Axis.Status.ErrorStop;
    _stAxis.stStatus.nErrorID := _stAxis.Axis.Status.ErrorID;//NC Error ID
ELSIF fbErrorRTrig.Q THEN
        //For each mcStatus
        FOR i := 1 TO nMCSTATUS_ARRAY_SIZE DO
            //If there's an error present propagate
            IF astMcStatus[i]^.ErrorID <> 0 THEN
                _stAxis.stStatus.nErrorID := astMcStatus[i]^.ErrorID;
            END_IF
        END_FOR
END_IF
END_METHOD

METHOD mStatus_InVelocity : BOOL
VAR
    i: UINT;
    tmpInVelocity: BOOL;
END_VAR
FOR i := 1 TO nMCSTATUS_ARRAY_SIZE DO
    tmpInVelocity := astMcStatus[i]^.InVelocity OR tmpInVelocity;
END_FOR
//fbInVelocityRTrig(CLK:= mStatus_InVelocity());
fbInVelocityRTrig(CLK := tmpInVelocity);
IF fbInVelocityRTrig.Q THEN
    _stAxis.stStatus.bInVelocity := TRUE;
END_IF

fbInVelocityFTrig(CLK := _stAxis.Axis.Status.ContinuousMotion);
IF fbInVelocityFTrig.Q THEN
    _stAxis.stStatus.bInVelocity := FALSE;
END_IF
END_METHOD

METHOD mStatus_MultiGearing : BOOL

IF _stAxis.Axis.Status.Coupled AND _stAxis.Axis.PlcToNc.GearRatio1 <> 0 AND _stAxis.stConfig.astMultiMasterAxisLatched[1].nIndex <> 0 THEN
    GVL.astAxes[_stAxis.stConfig.astMultiMasterAxisLatched[1].nIndex].stConfig.afMultiSlaveAxisRatio[GVL.iAxis] := _stAxis.Axis.PlcToNc.GearRatio1;
    _stAxis.stStatus.bCoupledGear1 := TRUE;
ELSE
    _stAxis.stStatus.bCoupledGear1 := FALSE;
END_IF

IF _stAxis.Axis.Status.Coupled AND _stAxis.Axis.PlcToNc.GearRatio2 <> 0 AND _stAxis.stConfig.astMultiMasterAxisLatched[2].nIndex <> 0 THEN
    GVL.astAxes[_stAxis.stConfig.astMultiMasterAxisLatched[2].nIndex].stConfig.afMultiSlaveAxisRatio[GVL.iAxis] := _stAxis.Axis.PlcToNc.GearRatio2;
    _stAxis.stStatus.bCoupledGear2 := TRUE;
ELSE
    _stAxis.stStatus.bCoupledGear2 := FALSE;
END_IF

IF _stAxis.Axis.Status.Coupled AND _stAxis.Axis.PlcToNc.GearRatio3 <> 0 AND _stAxis.stConfig.astMultiMasterAxisLatched[3].nIndex <> 0 THEN
    GVL.astAxes[_stAxis.stConfig.astMultiMasterAxisLatched[3].nIndex].stConfig.afMultiSlaveAxisRatio[GVL.iAxis] := _stAxis.Axis.PlcToNc.GearRatio3;
    _stAxis.stStatus.bCoupledGear3 := TRUE;
ELSE
    _stAxis.stStatus.bCoupledGear3 := FALSE;
END_IF

IF _stAxis.Axis.Status.Coupled AND _stAxis.Axis.PlcToNc.GearRatio4 <> 0 AND _stAxis.stConfig.astMultiMasterAxisLatched[4].nIndex <> 0 THEN
    GVL.astAxes[_stAxis.stConfig.astMultiMasterAxisLatched[4].nIndex].stConfig.afMultiSlaveAxisRatio[GVL.iAxis] := _stAxis.Axis.PlcToNc.GearRatio4;
    _stAxis.stStatus.bCoupledGear4 := TRUE;
ELSE
    _stAxis.stStatus.bCoupledGear4 := FALSE;
END_IF
END_METHOD

METHOD mStatus_NewCommand : BOOL
VAR
    i: UINT;
END_VAR

fbExecuteRTrig(CLK := _stAxis.stControl.bExecute);
IF fbExecuteRTrig.Q THEN
    _stAxis.stStatus.bDone := FALSE;
    _stAxis.stStatus.bCommandAborted := FALSE;

    //On a new motion command, clear the errorID
    CASE _stAxis.stControl.eCommand OF
            E_MotionFunctions.eMoveAbsolute,
            E_MotionFunctions.eMoveRelative,
            E_MotionFunctions.eMoveVelocity,
            E_MotionFunctions.eMoveModulo,
            E_MotionFunctions.eGearInMultiMaster,
            E_MotionFunctions.eGearOut,
            E_MotionFunctions.eHome :
                _stAxis.stStatus.nErrorID := 0;
            E_MotionFunctions.eWriteParameter,
            E_MotionFunctions.eReadParameter :
            // Nothing
    END_CASE
END_IF
END_METHOD

METHOD mStatus_Safety : BOOL
VAR
	iterator : UINT := 1;
	bTrippedPH : BOOL := FALSE;
END_VAR
(*
IF GVL_Safety.nSAFETY_OUTPUTS>0 THEN
	FOR iterator := 1 TO GVL_Safety.nSAFETY_OUTPUTS DO
		IF stSafetyData.aSafetyOuputs[iterator].abLinkedAxes[GVL.iAxis] THEN
			bTrippedPH := bTrippedPH OR stSafetyData.aSafetyOuputs[iterator].bTripped;
		END_IF
	END_FOR
END_IF

_stAxis.stSafety.bTripped := bTrippedPH;
*)
END_METHOD

METHOD Run : BOOL

mStatus_AxisStatus();
mParameters_ReadNc();
mParameters_Init();
stMcStatusReadParameter := mParameters_ReadParameter();
stMcStatusWriteParameter := mParameters_WriteParameter();

mControl_LimitHitTimer();
mControl_LimitLinking();
stMcStatusPower := mControl_Power();

stMcStatusHalt := mMove_Halt();
stMcStatusStop := mMove_Stop();
stMcStatusReset := mControl_Reset();

stMcStatusMoveAbsolute := mMove_MoveAbsolute();
stMcStatusMoveRelative := mMove_MoveRelative();
stMcStatusMoveModulo := mMove_MoveModulo();
stMcStatusMoveVelocity := mMove_MoveVelocity();

stMcStatusGearInMultiMaster := mControl_GearInMultiMaster();
stMcStatusGearOut := mControl_GearOut();

stMcStatusHome := mControl_Home();

mStatus_NewCommand();
mStatus_Done();
mStatus_Error();
mStatus_InVelocity();
mStatus_CommandAborted();
_stAxis.stStatus.bBusy := mStatus_Busy();

EndOfCycle();
END_METHOD

PROPERTY stAxis : REFERENCE TO ST_AxisStruct
GET
stAxis REF= _stAxis;
END_GET
SET
_stAxis REF= stAxis;
END_SET
END_PROPERTY

END_FUNCTION_BLOCK

// ---- POUs/Application_Specific/Applications/PLC_SAFETY_LOGIC.TcPOU
PROGRAM PLC_SAFETY_LOGIC
VAR
    
    iCounter : UINT := 1;
    
    safetyAckTon : TON;
    
    localModeButton_Pressed AT %I* : BOOL;
    localModeTon : TON;
    
    unoccupiedTon : TON;
    unoccupiedTrig : R_TRIG;
    sTempString : STRING;
    bSafetyDevicesSetup : BOOL:= FALSE;
    
    EStop1_ChA AT %I* : BOOL;
    EStop1_ChB AT %I* : BOOL;
    EStop2_ChA AT %I* : BOOL;
    EStop2_ChB AT %I* : BOOL;
    EStop3_ChA AT %I* : BOOL;
    EStop3_ChB AT %I* : BOOL;
    EStop4_ChA AT %I* : BOOL;
    EStop4_ChB AT %I* : BOOL;
    EStop5_ChA AT %I* : BOOL;
    EStop5_ChB AT %I* : BOOL;
    EStop6_ChA AT %I* : BOOL;
    EStop6_ChB AT %I* : BOOL;
    EStop7_ChA AT %I* : BOOL;
    EStop7_ChB AT %I* : BOOL;
    LightCurtain_ChA AT %I* : BOOL;
    LightCurtain_ChB AT %I* : BOOL;
    
    
END_VAR

IF bSafetyDevicesSetup = FALSE THEN
    ACT_SetupSafetyDevices();
END_IF



GVL_Safety.stSafetyData.SafetyGroups[1].AckGroup:= GVL_Safety.SAFETY_ACK;
GVL_Safety.stSafetyData.SafetyGroups[2].AckGroup:= GVL_Safety.SAFETY_ACK;
GVL_Safety.stSafetyData.SafetyGroups[3].AckGroup:= GVL_Safety.SAFETY_ACK;

//Convert STATE byte data to enum

ACT_ConvertFBState();
ACT_ConvertState();
ACT_LoadDiagnosticString();
ACT_ErrorAckReq();

IF GVL_Safety.stSafetyData.bSafetyAckReq THEN
    sTempString:= CONCAT(STR1:= 'Error on ',STR2:= GVL_Safety.stSafetyData.sInError);
    sTempString:= CONCAT(STR1:= sTempString,STR2:= ' : ');
    sTempString:= CONCAT(STR1:= sTempString,STR2:= GVL_Safety.stSafetyData.sInErrorDiag);
    GVL_Safety.stSafetyData.sDiagMessageToUser:= sTempString;
ELSE
    GVL_Safety.stSafetyData.sDiagMessageToUser:= '';
END_IF


//Load Diagnostics



/////OLD CODE BELOW
//GVL_Safety.ErrorAck_MotionSafety := GVL_Safety.Safety_Ack;
//GVL_Safety.ErrorAck_MotionSafety_XRotAndZHor := GVL_Safety.Safety_Ack;
//GVL_Safety.ErrorAck_MotionSafety_Y1AndY2 := GVL_Safety.Safety_Ack;

safetyAckTon(IN:= GVL_Safety.Safety_Ack, PT:= T#500MS);

IF safetyAckTon.Q  THEN
    GVL_Safety.Safety_Ack:= FALSE;
END_IF

//State valid monitoring block
IF GVL_Safety.stSafetyData.aSafetyFBS[10].State = 1 THEN
    GVL_Safety.LocalMode_Disabled:= FALSE;
ELSE
    GVL_Safety.LocalMode_Disabled:= TRUE;
END_IF




IF localModeButton_Pressed THEN
    localModeTon.IN:= TRUE;
    localModeTon.PT:= T#1S;        
END_IF
IF localModeTon.Q THEN
    GVL_INTER.RESET_ALL:= TRUE;
    localModeTon.IN:= FALSE;
END_IF
localModeTon();

unoccupiedTrig(CLK:= GVL_Safety.UnoccupiedMode);
IF unoccupiedTrig.Q THEN
    unoccupiedTon.IN:= TRUE;
    unoccupiedTon.PT:= T#1S;
END_IF
IF unoccupiedTon.Q THEN
    GVL_INTER.RESET_ALL:= TRUE;
    unoccupiedTon.IN:= FALSE;
END_IF
unoccupiedTon();

ACTION ACT_ConvertFBState:
GVL_Safety.stSafetyData.bSafetyAckReq:= FALSE;
FOR iCounter:=1 TO GVL_Safety.nSAFETY_FBS DO
    GVL_Safety.stSafetyData.aSafetyFBS[iCounter].fbState:= USINT_TO_INT(GVL_Safety.stSafetyData.aSafetyFBS[iCounter].State); 
END_FOR
END_ACTION

ACTION ACT_ConvertState:

FOR iCounter:=1 TO GVL_Safety.nSAFETY_GROUPS DO
    GVL_Safety.stSafetyData.SafetyGroups[iCounter].groupState:= BYTE_TO_INT(GVL_Safety.stSafetyData.SafetyGroups[iCounter].Status); 
END_FOR
END_ACTION

ACTION ACT_ErrorAckReq:
GVL_Safety.stSafetyData.bSafetyAckReq:= FALSE;
FOR iCounter:=1 TO GVL_Safety.nSAFETY_GROUPS DO
    IF GVL_Safety.stSafetyData.SafetyGroups[iCounter].groupState = E_SafetyGroupState.ERROR THEN
        GVL_Safety.stSafetyData.bSafetyAckReq:= TRUE;
       GVL_Safety.stSafetyData.sInError := GVL_Safety.stSafetyData.SafetyGroups[iCounter].Name;
	END_IF
END_FOR

FOR iCounter:=1 TO GVL_Safety.nSAFETY_FBS DO
    IF GVL_Safety.stSafetyData.aSafetyFBS[iCounter].fbState = E_SafetyFbState.ERROR THEN
        GVL_Safety.stSafetyData.bSafetyAckReq:= TRUE;
        GVL_Safety.stSafetyData.sInError := GVL_Safety.stSafetyData.aSafetyFBS[iCounter].sName;
        GVL_Safety.stSafetyData.sInErrorDiag := GVL_Safety.stSafetyData.aSafetyFBS[iCounter].DiagString;
	END_IF
END_FOR
END_ACTION

ACTION ACT_LoadDiagnosticString:
FOR iCounter:=1 TO GVL_Safety.nSAFETY_FBS DO
    IF GVL_Safety.stSafetyData.aSafetyFBS[iCounter].State=4 THEN
        GVL_Safety.stSafetyData.aSafetyFBS[iCounter].DiagString:= FB_SafeFBDiag(
        fbType:= GVL_Safety.stSafetyData.aSafetyFBS[iCounter].eFbType,
        diagVal:= GVL_Safety.stSafetyData.aSafetyFBS[iCounter].Diag);
	ELSE
        GVL_Safety.stSafetyData.aSafetyFBS[iCounter].DiagString:='';
    END_IF
    

END_FOR
END_ACTION

ACTION ACT_SetupSafetyDevices:
//DO ALL STRING AND TYPE SETUP HERE
GVL_Safety.stSafetyData.SafetyGroups[1].Name:= 'EL6910';
GVL_Safety.stSafetyData.SafetyGroups[2].Name:= 'XRot and ZTrans - AXdrives';
GVL_Safety.stSafetyData.SafetyGroups[3].Name:= 'Y1 and Y2 - AXdrives';

GVL_Safety.stSafetyData.aSafetyFBS[1].sName:= 'FB_Mon - Lightcurtain';
GVL_Safety.stSafetyData.aSafetyFBS[1].eFbType:= E_SafetyFbType.FB_Mon;

GVL_Safety.stSafetyData.aSafetyFBS[2].sName:= 'FB_Mon - SearchedAndLocked';
GVL_Safety.stSafetyData.aSafetyFBS[2].eFbType:= E_SafetyFbType.FB_Mon;

GVL_Safety.stSafetyData.aSafetyFBS[3].sName:= 'FB_Mon - LocalModeDisable';
GVL_Safety.stSafetyData.aSafetyFBS[3].eFbType:= E_SafetyFbType.FB_Mon;

GVL_Safety.stSafetyData.aSafetyFBS[4].sName:= 'FB_OpMode - OpMode';
GVL_Safety.stSafetyData.aSafetyFBS[4].eFbType:= E_SafetyFbType.FB_OpMode;

GVL_Safety.stSafetyData.aSafetyFBS[5].sName:= 'FB_Mon - EStopsCloche';
GVL_Safety.stSafetyData.aSafetyFBS[5].eFbType:= E_SafetyFbType.FB_Mon;

GVL_Safety.stSafetyData.aSafetyFBS[6].sName:= 'FB_Mon - EStopsSample';
GVL_Safety.stSafetyData.aSafetyFBS[6].eFbType:= E_SafetyFbType.FB_Mon;

GVL_Safety.stSafetyData.aSafetyFBS[7].sName:= 'FB_Mon - EStopsRear';
GVL_Safety.stSafetyData.aSafetyFBS[7].eFbType:= E_SafetyFbType.FB_Mon;

GVL_Safety.stSafetyData.aSafetyFBS[8].sName:= 'FB_Mon - EStopsPanel';
GVL_Safety.stSafetyData.aSafetyFBS[8].eFbType:= E_SafetyFbType.FB_Mon;

GVL_Safety.stSafetyData.aSafetyFBS[9].sName:= 'FB_Mon - EStopsCombined';
GVL_Safety.stSafetyData.aSafetyFBS[9].eFbType:= E_SafetyFbType.FB_Mon;

GVL_Safety.stSafetyData.aSafetyFBS[10].sName:= 'FB_Mon - StateValid';
GVL_Safety.stSafetyData.aSafetyFBS[10].eFbType:= E_SafetyFbType.FB_Mon;

GVL_Safety.stSafetyData.aSafetyFBS[11].sName:= 'FB_RS - ResetToAxDrives';
GVL_Safety.stSafetyData.aSafetyFBS[11].eFbType:= E_SafetyFbType.FB_RS;

GVL_Safety.stSafetyData.aSafetyFBS[12].sName:= 'FB_EDM - BeckhoffContactor';
GVL_Safety.stSafetyData.aSafetyFBS[12].eFbType:= E_SafetyFbType.FB_EDM;

GVL_Safety.stSafetyData.aSafetyFBS[13].sName:= 'FB_EDM - GalilContactor';
GVL_Safety.stSafetyData.aSafetyFBS[13].eFbType:= E_SafetyFbType.FB_EDM;

GVL_Safety.stSafetyData.aSafetyFBS[14].sName:= 'FB_EDM - RotationBrake1';
GVL_Safety.stSafetyData.aSafetyFBS[14].eFbType:= E_SafetyFbType.FB_EDM;

GVL_Safety.stSafetyData.aSafetyFBS[15].sName:= 'FB_EDM - RotationBrake2';
GVL_Safety.stSafetyData.aSafetyFBS[15].eFbType:= E_SafetyFbType.FB_EDM;







bSafetyDevicesSetup:= TRUE;
END_ACTION

END_PROGRAM

// ---- tc_mca_std_lib/DUTs/Safety Status/FB_SafeFBDiag.TcPOU
FUNCTION FB_SafeFBDiag : STRING
VAR_INPUT
    fbType : E_SafetyFbType;
    diagVal : UINT;
END_VAR
VAR
    diagnosticMessage : STRING;
END_VAR

CASE fbType OF
    E_SafetyFbType.FB_Mon:
        IF diagVal.0 THEN
            diagnosticMessage:= 'Discrepancy error input group 1';
		ELSIF diagVal.1 THEN        
            diagnosticMessage:= 'Discrepancy error input group 2';
        ELSIF diagVal.2 THEN
                diagnosticMessage:= 'Discrepancy error in Secure input group';
        ELSIF diagVal.4 THEN
                diagnosticMessage:= 'EDM monitoring error EDM1';
        ELSIF diagVal.5 THEN
                diagnosticMessage:= 'EDM monitoring error EDM2';
        ELSIF diagVal.8 THEN
                diagnosticMessage:= 'Discrepancy error input group 1';
        ELSIF diagVal.9 THEN
                diagnosticMessage:= 'Discrepancy error input group 2';
        ELSIF diagVal.10 THEN
                diagnosticMessage:= 'Discrepancy error input group Secure';
        ELSE
                diagnosticMessage:= ' ';
		END_IF
   ELSE
       diagnosticMessage:='';
END_CASE

FB_SafeFBDiag:= diagnosticMessage;

END_FUNCTION

// ---- POUs/Application_Specific/Axes/Horizontal_Translation.TcPOU
PROGRAM Horizontal_Translation
VAR
//Outputs: Power for Limit switches, Home Sensors, etc.
    bFwdLimitPower AT %Q* : BOOL := TRUE;
    bBwdLimitPower AT %Q* : BOOL := TRUE;
    bEnable : BOOL :=TRUE;
    //bPowerSwitchesAxis1 AT %Q*: BOOL:= TRUE;

//Hardware interlocks
    //bInterlockFwdOK AT %I*: BOOL;
END_VAR

//Initial parameters of an Axis
IF _TaskInfo[fbGetCurTaskIndex.index].FirstCycle THEN
    //Initial default values:
    //Absolute encoder
    GVL.astAxes[AXIS_HORIZONTAL_TRANSLATION].stConfig.eHomeSeq := E_HomingRoutines.eNoHoming;
    //GVL.astAxes[1].stConfig.fHomePosition := 0.0;
    //GVL.astAxes[1].stConfig.fHomeFinishDistance := 0.0;
    //GVL.astAxes[1].stConfig.eRestorePosition := E_RestorePosition.eRestoreWithoutHome;
END_IF

astAxes[AXIS_HORIZONTAL_TRANSLATION].stControl.bEnable := bEnable;
astAxes[AXIS_HORIZONTAL_TRANSLATION].stDescription.sAxisName := 'HORIZ_TRANSL';
//Define ACTIONS() or write exclusive code for an specific axis.
(*Eg. Stop when temperature reaches certain values, reduce speed if  a signal is activated, etc.
Eg. GVL.astAxes[x].stControl.bInterlockFwd := NOT bInterlockFwdOK;*)

END_PROGRAM

// ---- POUs/Application_Specific/Axes/Vertical_Translation_Y2.TcPOU
PROGRAM Vertical_Translation_Y2
VAR
//Outputs: Power for Limit switches, Home Sensors, etc.
    bFwdLimitPower AT %Q* : BOOL := TRUE;
    bBwdLimitPower AT %Q* : BOOL := TRUE;
    //bPowerSwitchesAxis1 AT %Q*: BOOL:= TRUE;

//Hardware interlocks
    //bInterlockFwdOK AT %I*: BOOL;
END_VAR

//Initial parameters of an Axis
(*IF _TaskInfo[fbGetCurTaskIndex.index].FirstCycle THEN
    //Initial default values:
    GVL.astAxes[1].stConfig.eHomeSeq := 0;
    GVL.astAxes[1].stConfig.fHomePosition := 0.0;
    GVL.astAxes[1].stConfig.fHomeFinishDistance := 0.0;
    GVL.astAxes[1].stConfig.eRestorePosition := E_RestorePosition.eRestoreWithoutHome;
END_IF*)

astAxes[AXIS_VERTICAL_TRANSLATION_Y2].stControl.bEnable := TRUE;
astAxes[AXIS_VERTICAL_TRANSLATION_Y2].stDescription.sAxisName := 'VERT_Y2';
//Define ACTIONS() or write exclusive code for an specific axis.
(*Eg. Stop when temperature reaches certain values, reduce speed if  a signal is activated, etc.
Eg. GVL.astAxes[x].stControl.bInterlockFwd := NOT bInterlockFwdOK;*)

END_PROGRAM

// ---- POUs/Application_Specific/Axes/Vertical_Translation_Y1.TcPOU
PROGRAM Vertical_Translation_Y1
VAR
//Outputs: Power for Limit switches, Home Sensors, etc.
    //bPowerSwitchesAxis1 AT %Q*: BOOL:= TRUE;
    bFwdLimitPower AT %Q* : BOOL := TRUE;
    bBwdLimitPower AT %Q* : BOOL := TRUE;
//Hardware interlocks
    //bInterlockFwdOK AT %I*: BOOL;
END_VAR

//Initial parameters of an Axis
(*IF _TaskInfo[fbGetCurTaskIndex.index].FirstCycle THEN
    //Initial default values:
    GVL.astAxes[1].stConfig.eHomeSeq := 0;
    GVL.astAxes[1].stConfig.fHomePosition := 0.0;
    GVL.astAxes[1].stConfig.fHomeFinishDistance := 0.0;
    GVL.astAxes[1].stConfig.eRestorePosition := E_RestorePosition.eRestoreWithoutHome;
END_IF*)

astAxes[AXIS_VERTICAL_TRANSLATION_Y1].stControl.bEnable := TRUE;
astAxes[AXIS_VERTICAL_TRANSLATION_Y1].stDescription.sAxisName := 'VERT_Y1';
//Define ACTIONS() or write exclusive code for an specific axis.
(*Eg. Stop when temperature reaches certain values, reduce speed if  a signal is activated, etc.
Eg. GVL.astAxes[x].stControl.bInterlockFwd := NOT bInterlockFwdOK;*)

END_PROGRAM

// ---- POUs/Application_Specific/Axes/Rotation.TcPOU
PROGRAM Rotation
VAR
//Outputs: Power for Limit switches, Home Sensors, etc.
    //bPowerSwitchesAxis1 AT %Q*: BOOL:= TRUE;
    bFwdLimitPower AT %Q* : BOOL := TRUE;
    bBwdLimitPower AT %Q* : BOOL := TRUE;
    bEnable : BOOL := TRUE;
    
    OpState : E_RotationBrakeCheckerState := E_RotationBrakeCheckerState.init;
    OpSate_String : STRING;
    bBrakeTestInProgress : BOOL;
    fbBrakeControl : FB_CoEAX8000BrakeControl;
    
    fbReadDriveOpMode : MC_ReadDriveOperationMode;
    driveOpModeReadIn : E_DriveOperationMode;
    sErrorMessage : STRING;
    bInBrakeTestMode AT %I* : BOOL;
    
    Brake1Valid AT %I* : BOOL;
    Brake1State AT %I* : BOOL;
    Brake2Valid AT %I* : BOOL;
    Brake2State AT %I* : BOOL;
    
    TriggerBrake1Test : BOOL; //PLC test trigger
    TriggerBrake2Test : BOOL; //PLC test trigger
    
    RunBrake1Test AT %Q* : BOOL; // Test trigger to safety system
    RunBrake2Test AT %Q* : BOOL; // Test trigger to safety system
    TestingBrake1 : BOOL;
    TestingBrake2 : BOOL;
    FinishBrakeTesting AT %Q* : BOOL;
    ManualReleaseBrake1 AT %Q* : BOOL;
    ManualReleaseBrake2 AT %Q* : BOOL;
    RotationSTOState AT %I* : BOOL;
    Reinitialise : BOOL; //Bool to get out of error state
    
    Brake1TimeRemaining_RAW AT %I* : UDINT; //In seconds
    Brake2TimeRemaining_RAW AT %I* : UDINT; //In seconds
    Brake1TimeRemaining_Breakdown : UDINT;
    Brake2TimeRemaining_Breakdown : UDINT;
    
    Brake1TimeRemaining_Days : UDINT;
    Brake1TimeRemaining_Hours : UDINT;
    Brake1TimeRemaining_Minutes : UDINT;
    Brake1TimeRemaining_Seconds : UDINT;
    
    
    Brake2TimeRemaining_Days : UDINT;
    Brake2TimeRemaining_Hours : UDINT;
    Brake2TimeRemaining_Minutes : UDINT;
    Brake2TimeRemaining_Seconds : UDINT;
    
    iQ_Current AT %I* : REAL;
    SBC_FailsafeFault AT %I* : BOOL;
    BC1_Error AT %I* : BOOL;
    BC2_Error AT %I* : BOOL;
    BrakeReset AT %Q* : BOOL;
    
    
    stateTimout : TON;
    brakeDelay : TON;
    loadDelay : TON;
    timeToClearValid : TON;
    brakeResetTon : TON;
    
    fbAx8000BrakeTest : FB_CoEAX8000BrakeTest;
    fbReset : MC_Reset();
    
    TEST_TORQUE : LREAL := 2.1;//1.4142;
    ResetCounter : INT;
    ResetCounterLimit : INT := 5;
//Hardware interlocks
    //bInterlockFwdOK AT %I*: BOOL;
END_VAR
VAR CONSTANT
    DAY_SECONDS : UDINT := 86400;
    HOUR_SECONDS : UDINT := 3600;
    MINUTE_SECONDS : UDINT := 60;
END_VAR

OpSate_String := TO_STRING(OpState);
brakeResetTon(IN:=BrakeReset, PT:=T#250MS);
IF brakeResetTon.Q THEN
    BrakeReset:= FALSE;
END_IF

//Time conversion logic
Brake1TimeRemaining_Days:= Brake1TimeRemaining_RAW/DAY_SECONDS;
Brake1TimeRemaining_Breakdown := Brake1TimeRemaining_RAW MOD DAY_SECONDS;
Brake1TimeRemaining_Hours:= Brake1TimeRemaining_Breakdown/HOUR_SECONDS;
Brake1TimeRemaining_Breakdown:= Brake1TimeRemaining_Breakdown MOD HOUR_SECONDS;
Brake1TimeRemaining_Minutes:= Brake1TimeRemaining_Breakdown/MINUTE_SECONDS;
Brake1TimeRemaining_Breakdown:= Brake1TimeRemaining_Breakdown MOD MINUTE_SECONDS;
Brake1TimeRemaining_Seconds:= Brake1TimeRemaining_Breakdown;

Brake2TimeRemaining_Days:= Brake2TimeRemaining_RAW/DAY_SECONDS;
Brake2TimeRemaining_Breakdown := Brake2TimeRemaining_RAW MOD DAY_SECONDS;
Brake2TimeRemaining_Hours:= Brake2TimeRemaining_Breakdown/HOUR_SECONDS;
Brake2TimeRemaining_Breakdown:= Brake2TimeRemaining_Breakdown MOD HOUR_SECONDS;
Brake2TimeRemaining_Minutes:= Brake2TimeRemaining_Breakdown/MINUTE_SECONDS;
Brake2TimeRemaining_Breakdown:= Brake2TimeRemaining_Breakdown MOD MINUTE_SECONDS;
Brake2TimeRemaining_Seconds:= Brake2TimeRemaining_Breakdown;

//Actual brake logic
GVL_INTER.BRAKE_TEST_PASSED:= Brake1Valid AND Brake2Valid; //Feedback from safety system as to if brake test is passed

astAxes[AXIS_ROTATION].stControl.bEnable := FALSE;  //Will be overridden by state machine
astAxes[AXIS_ROTATION].stDescription.sAxisName := 'ROTATION';


IF NOT GVL_INTER.BRAKE_TEST_PASSED AND NOT bBrakeTestInProgress THEN
    OpState:= E_RotationBrakeCheckerState.init;
END_IF

CASE OpState OF
    E_RotationBrakeCheckerState.init:
        //Ensure motor cannot be enabled
        bBrakeTestInProgress:=FALSE;
        FinishBrakeTesting:=FALSE;
        
        //Ensure no "active brake test signals"
        RunBrake1Test:= FALSE;
        RunBrake2Test:= FALSE;
        ManualReleaseBrake1:=FALSE;
        ManualReleaseBrake2:=FALSE;
        IF GVL_INTER.BRAKE_TEST_PASSED THEN
            OpState:= E_RotationBrakeCheckerState.Set_Brake_Mode_To_Op;
        END_IF
        IF bInBrakeTestMode THEN
            bBrakeTestInProgress:= TRUE;
            OpState:= E_RotationBrakeCheckerState.Start_Brake_Test;            
		END_IF
    
    E_RotationBrakeCheckerState.Set_Brake_Mode_To_Op:
        fbBrakeControl.Execute:= TRUE;
        fbBrakeControl.Mode:= E_AX8000BrakeMode.eAX8000BrakeMode_Automatic;
        fbBrakeControl(Axis:= astAxes[AXIS_ROTATION].Axis);
        OpState:= E_RotationBrakeCheckerState.Check_Brake_Mode_To_Op;
    
    E_RotationBrakeCheckerState.Check_Brake_Mode_To_Op:
        fbBrakeControl(Axis:= astAxes[AXIS_ROTATION].Axis); //Run function block to update statuses    
        IF NOT fbBrakeControl.Busy AND NOT fbBrakeControl.Error THEN
            fbBrakeControl.Execute:= FALSE;
            fbBrakeControl.Mode:= E_AX8000BrakeMode.eAX8000BrakeMode_Automatic;
            fbBrakeControl(Axis:= astAxes[AXIS_ROTATION].Axis);
            OpState:= E_RotationBrakeCheckerState.Check_Drive_Mode_To_Op;
        ELSIF NOT fbBrakeControl.Busy AND fbBrakeControl.Error THEN
            fbBrakeControl.Execute:= FALSE;
            fbBrakeControl.Mode:= E_AX8000BrakeMode.eAX8000BrakeMode_Automatic;
            fbBrakeControl(Axis:= astAxes[AXIS_ROTATION].Axis);
            OpState:= E_RotationBrakeCheckerState.Error;
            sErrorMessage:= 'Unable to set brake mode to automatic whilst moving to inop';
        END_IF
        
    E_RotationBrakeCheckerState.Check_Drive_Mode_To_Op:
        fbReadDriveOpMode(Axis:= astAxes[AXIS_ROTATION].Axis,Execute:= TRUE);
        
        IF NOT fbReadDriveOpMode.Busy AND NOT fbReadDriveOpMode.Error THEN
            driveOpModeReadIn := fbReadDriveOpMode.DriveOperationMode;
            fbReadDriveOpMode(Axis:= astAxes[AXIS_ROTATION].Axis,Execute:= FALSE);
            IF driveOpModeReadIn = E_DriveOperationMode.DriveOperationMode_Pos1 OR driveOpModeReadIn = E_DriveOperationMode.DriveOperationMode_Default THEN
                OpState:= E_RotationBrakeCheckerState.In_Operation;
            ELSE
                OpState:= E_RotationBrakeCheckerState.Error;
                sErrorMessage:= 'Incorrect drive op mode when moving to InOp';
			END_IF
		END_IF
        IF NOT fbReadDriveOpMode.Busy AND fbReadDriveOpMode.Error THEN
            fbReadDriveOpMode(Axis:= astAxes[AXIS_ROTATION].Axis,Execute:= FALSE);
            OpState:= E_RotationBrakeCheckerState.Error;
            sErrorMessage:= 'Error reading drive operation mode';
		END_IF
        
     E_RotationBrakeCheckerState.In_Operation:
        //DO NOTHING
        ManualReleaseBrake1:=TRUE;
        ManualReleaseBrake2:=TRUE;
        astAxes[AXIS_ROTATION].stControl.bEnable := bEnable;
        
        IF NOT GVL_INTER.BRAKE_TEST_PASSED OR bInBrakeTestMode THEN
            OpState:= E_RotationBrakeCheckerState.init;
		END_IF
        
     E_RotationBrakeCheckerState.Error:
        ManualReleaseBrake1:= FALSE;
        ManualReleaseBrake2:= FALSE;
        ResetCounter:= 0;
        IF Reinitialise THEN
            OpState:= E_RotationBrakeCheckerState.init;
		END_IF
        
    //////////BRAKE TESTING SEQUENCE ////////
    E_RotationBrakeCheckerState.Start_Brake_Test:
        astAxes[AXIS_ROTATION].stControl.bEnable := FALSE;
        //Confirm brakes are on and unlock AX motor brake
        //Remember, to test brake 1, you must release brake 2!!!
        ManualReleaseBrake1:= FALSE;
        ManualReleaseBrake2:= FALSE;
        
        //Brakes are not on (holding)
        IF NOT Brake1State AND NOT Brake2State THEN
            //Release ax motor brake
            fbBrakeControl.Execute:= TRUE;
            fbBrakeControl.Mode:= E_AX8000BrakeMode.eAX8000BrakeMode_Unlock;
            fbBrakeControl(Axis:= astAxes[AXIS_ROTATION].Axis);
            
            IF NOT fbBrakeControl.Busy AND NOT fbBrakeControl.Error THEN
                fbBrakeControl.Execute:= FALSE;
                fbBrakeControl.Mode:= E_AX8000BrakeMode.eAX8000BrakeMode_Unlock;
                fbBrakeControl(Axis:= astAxes[AXIS_ROTATION].Axis);
                OpState:= E_RotationBrakeCheckerState.Reset_Axis;
            ELSIF NOT fbBrakeControl.Busy AND fbBrakeControl.Error THEN
                fbBrakeControl.Execute:= FALSE;
                fbBrakeControl.Mode:= E_AX8000BrakeMode.eAX8000BrakeMode_Automatic;
                fbBrakeControl(Axis:= astAxes[AXIS_ROTATION].Axis);
                OpState:= E_RotationBrakeCheckerState.Error;
                sErrorMessage:= 'Unable to set brake mode to automatic whilst performing brake test';
            END_IF
            
		END_IF
        
        E_RotationBrakeCheckerState.Reset_Axis:
        //NEED TO DO MY OWN RESET LOGIC HERE - WAS IN ERROR STATE
            astAxes[AXIS_ROTATION].stControl.bEnable := FALSE;
            ManualReleaseBrake1:= FALSE;
            ManualReleaseBrake2:= FALSE;
            astAxes[AXIS_ROTATION].stControl.bReset:= TRUE;
            
            stateTimout(IN:= TRUE, PT:=T#2S);
            GVL_INTER.RESET_ALL:= TRUE;
            //If no error
            IF NOT astAxes[AXIS_ROTATION].Axis.Status.Error THEN
                stateTimout(IN:= FALSE);
                OpState:= E_RotationBrakeCheckerState.Confirm_STO_State;
			END_IF
            IF stateTimout.Q THEN
                stateTimout(IN:= FALSE);
                OpState:= E_RotationBrakeCheckerState.Error;
                sErrorMessage:= 'Unable to reset axis error';
			END_IF
            
        E_RotationBrakeCheckerState.Confirm_STO_State:
            astAxes[AXIS_ROTATION].stControl.bEnable := FALSE;
            ManualReleaseBrake1:= FALSE;
            ManualReleaseBrake2:= FALSE;
            stateTimout(IN:= TRUE, PT:=T#2S);
            IF NOT RotationSTOState THEN
                stateTimout(IN:= FALSE);
                OpState:= E_RotationBrakeCheckerState.Enable_Motor;
			END_IF
            IF stateTimout.Q THEN
                stateTimout(IN:= FALSE);
                OpState:= E_RotationBrakeCheckerState.Error;
                sErrorMessage:= 'AXIS STO';
			END_IF
            
        E_RotationBrakeCheckerState.Enable_Motor:
            ManualReleaseBrake1:= FALSE;
            ManualReleaseBrake2:= FALSE;
            stateTimout(IN:= TRUE, PT:=T#2S);
            astAxes[AXIS_ROTATION].stControl.bEnable:= TRUE;
            
            IF astAxes[AXIS_ROTATION].stStatus.bEnabled THEN
                stateTimout(IN:= FALSE);
                OpState:= E_RotationBrakeCheckerState.Wait_For_Test_Trigger;
			END_IF
            IF stateTimout.Q THEN
                stateTimout(IN:= FALSE);
                OpState:= E_RotationBrakeCheckerState.Error;
                sErrorMessage:= 'Axis could not enable';
			END_IF
        
        E_RotationBrakeCheckerState.Wait_For_Test_Trigger:
            IF GVL.astAxes[AXIS_ROTATION].Axis.Status.Error THEN
                GVL_INTER.RESET_ALL:= TRUE;
                ResetCounter:= ResetCounter +1;
                IF ResetCounter>ResetCounterLimit THEN
                    OpState:= E_RotationBrakeCheckerState.Error;
                    sErrorMessage:= 'Axis in error state, cannot be reset';
                END_IF
			END_IF
            astAxes[AXIS_ROTATION].stControl.bEnable:= TRUE;
        //We have an enabled motor, brake mode unlocked, all errors cleared
            ManualReleaseBrake1:= FALSE;
            ManualReleaseBrake2:= FALSE;
            fbAx8000BrakeTest(Axis:= astAxes[AXIS_ROTATION].Axis,
                Execute:= FALSE);
            
            //Does not clear brake test mode (yet?)
            IF FinishBrakeTesting OR NOT bInBrakeTestMode THEN
                OpState:= E_RotationBrakeCheckerState.Finishing_Brake_Test;                
			END_IF
            TestingBrake1:= FALSE;
            TestingBrake2:= FALSE;
            RunBrake1Test:= FALSE;
            RunBrake2Test:= FALSE;
            
            IF TriggerBrake1Test THEN
                TestingBrake1:= TRUE;
                ManualReleaseBrake2:= TRUE;
                OpState:= E_RotationBrakeCheckerState.Brake_Disengage_Delay;
			END_IF
            IF TriggerBrake2Test THEN
                TestingBrake2:= TRUE;
                ManualReleaseBrake1:= TRUE;
                OpState:= E_RotationBrakeCheckerState.Brake_Disengage_Delay;
			END_IF
            
        E_RotationBrakeCheckerState.Brake_Disengage_Delay:
            astAxes[AXIS_ROTATION].stControl.bEnable:= TRUE;
            brakeDelay(IN:= TRUE, PT:=T#1000MS);
            
            //Brake 1 tester
            IF TestingBrake1 AND Brake2State AND brakeDelay.Q THEN
                brakeDelay(IN:= FALSE);
                OpState:= E_RotationBrakeCheckerState.Brake_Test_Triggered;
			END_IF
            
            //Brake 2 tester
            IF TestingBrake2 AND Brake1State AND brakeDelay.Q THEN
                brakeDelay(IN:= FALSE);
                OpState:= E_RotationBrakeCheckerState.Brake_Test_Triggered;
			END_IF
            
        E_RotationBrakeCheckerState.Brake_Test_Triggered:
            astAxes[AXIS_ROTATION].stControl.bEnable:= TRUE;
            loadDelay(IN:= TRUE, PT:=T#500MS);
            timeToClearValid(IN:= TRUE, PT:=T#750MS);
            IF TestingBrake2 THEN
                IF loadDelay.Q THEN
                    RunBrake2Test := TRUE;
				END_IF               
                ManualReleaseBrake2:= FALSE;                
			END_IF
            IF TestingBrake1 THEN
                IF loadDelay.Q THEN
                    RunBrake1Test := TRUE;
				END_IF
                ManualReleaseBrake1:= FALSE;                
			END_IF
            fbAx8000BrakeTest(Axis:= astAxes[AXIS_ROTATION].Axis,
                Execute:= TRUE, 
                Torque:= TEST_TORQUE, 
                VelocityLimit:= 10,
                Succeeded:=FALSE,
                Timeout:= T#10S);
            
            IF timeToClearValid.Q THEN
                loadDelay(IN:= FALSE, PT:=T#500MS);
                timeToClearValid(IN:= FALSE, PT:=T#750MS);
                OpState:= E_RotationBrakeCheckerState.Brake_Testing_Underway;
			END_IF
            
        E_RotationBrakeCheckerState.Brake_Testing_Underway:
            astAxes[AXIS_ROTATION].stControl.bEnable:= TRUE;
            //Ensure only 1 brake released
            IF TestingBrake1 THEN
                fbAx8000BrakeTest.Succeeded:= Brake1Valid;
            ELSIF TestingBrake2 THEN
                fbAx8000BrakeTest.Succeeded:= Brake2Valid;
			END_IF
            
            fbAx8000BrakeTest(Axis:= astAxes[AXIS_ROTATION].Axis,
                Execute:= TRUE);

           IF NOT fbAx8000BrakeTest.Busy AND NOT fbAx8000BrakeTest.Error THEN
               fbAx8000BrakeTest(Axis:= astAxes[AXIS_ROTATION].Axis, Execute:= FALSE);
               OpState:= E_RotationBrakeCheckerState.Wait_For_Test_Trigger;
               RunBrake1Test:=FALSE;
               RunBrake2Test:=FALSE;
               TriggerBrake1Test:= FALSE;
               TriggerBrake2Test:= FALSE;
               loadDelay(IN:= FALSE, PT:=T#500MS);
		   ELSIF NOT fbAx8000BrakeTest.Busy AND fbAx8000BrakeTest.Error THEN
               fbAx8000BrakeTest(Axis:= astAxes[AXIS_ROTATION].Axis, Execute:= FALSE);
               OpState:= E_RotationBrakeCheckerState.Wait_For_Test_Trigger;
               RunBrake1Test:=FALSE;
               RunBrake2Test:=FALSE;
               TriggerBrake1Test:= FALSE;
               TriggerBrake2Test:= FALSE;
               loadDelay(IN:= FALSE, PT:=T#500MS);
            END_IF
        
        E_RotationBrakeCheckerState.Finishing_Brake_Test:
            ManualReleaseBrake1:= FALSE;
            ManualReleaseBrake2:= FALSE;
            
            fbBrakeControl.Execute:= TRUE;
            fbBrakeControl.Mode:= E_AX8000BrakeMode.eAX8000BrakeMode_Automatic;
            fbBrakeControl(Axis:= astAxes[AXIS_ROTATION].Axis);
            
            IF NOT fbBrakeControl.Busy AND NOT fbBrakeControl.Error THEN
                fbBrakeControl.Execute:= FALSE;
                fbBrakeControl.Mode:= E_AX8000BrakeMode.eAX8000BrakeMode_Automatic;
                fbBrakeControl(Axis:= astAxes[AXIS_ROTATION].Axis);
                OpState:= E_RotationBrakeCheckerState.init;
            ELSIF NOT fbBrakeControl.Busy AND fbBrakeControl.Error THEN
                fbBrakeControl.Execute:= FALSE;
                fbBrakeControl.Mode:= E_AX8000BrakeMode.eAX8000BrakeMode_Automatic;
                fbBrakeControl(Axis:= astAxes[AXIS_ROTATION].Axis);
                OpState:= E_RotationBrakeCheckerState.Error;
                sErrorMessage:= 'Unable to set brake mode to automatic whilst performing brake test';
            END_IF
END_CASE
Reinitialise:= FALSE;

END_PROGRAM

// ---- POUs/Application_Specific/Axes/Combined_Vertical.TcPOU
PROGRAM Combined_Vertical
VAR
//Outputs: Power for Limit switches, Home Sensors, etc.
    //bPowerSwitchesAxis1 AT %Q*: BOOL:= TRUE;

//Hardware interlocks
    //bInterlockFwdOK AT %I*: BOOL;
END_VAR

//Initial parameters of an Axis
(*IF _TaskInfo[fbGetCurTaskIndex.index].FirstCycle THEN
    //Initial default values:
    GVL.astAxes[1].stConfig.eHomeSeq := 0;
    GVL.astAxes[1].stConfig.fHomePosition := 0.0;
    GVL.astAxes[1].stConfig.fHomeFinishDistance := 0.0;
    GVL.astAxes[1].stConfig.eRestorePosition := E_RestorePosition.eRestoreWithoutHome;
END_IF*)
astAxes[AXIS_COMBINED_VERTICAL].stInputs.bLimitFwd := astAxes[AXIS_VERTICAL_TRANSLATION_Y1].stInputs.bLimitFwd AND astAxes[AXIS_VERTICAL_TRANSLATION_Y2].stInputs.bLimitFwd;
astAxes[AXIS_COMBINED_VERTICAL].stInputs.bLimitBwd := astAxes[AXIS_VERTICAL_TRANSLATION_Y1].stInputs.bLimitBwd AND astAxes[AXIS_VERTICAL_TRANSLATION_Y2].stInputs.bLimitBwd;

astAxes[AXIS_COMBINED_VERTICAL].stDescription.sAxisName := 'COMBINED_Y';
//Define ACTIONS() or write exclusive code for an specific axis.
(*Eg. Stop when temperature reaches certain values, reduce speed if  a signal is activated, etc.
Eg. GVL.astAxes[x].stControl.bInterlockFwd := NOT bInterlockFwdOK;*)

//astAxes[AXIS_COMBINED_VERTICAL].stControl.bEnable := astAxes[AXIS_VERTICAL_TRANSLATION_Z1].stStatus.bEnabled AND astAxes[AXIS_VERTICAL_TRANSLATION_Z2].stStatus.bEnabled;
(*
This will be the axis that drives the vertical stages, there will be no "real master"
This axis will only be able to run if the two axes below it are coupled in.
*)

END_PROGRAM

// ---- POUs/Application_Specific/Axes/Virtuals/Drad_External.TcPOU
PROGRAM Drad_External
VAR
    fEncoderPosition : LREAL;
    EncoderPosition AT %Q* : DINT; //Encoder value for NC
    fScaler : LREAL := 100000;
END_VAR

astAxes[AXIS_DRAD_EXTERNAL].stInputs.bLimitBwd := TRUE;
astAxes[AXIS_DRAD_EXTERNAL].stInputs.bLimitFwd := TRUE;
astAxes[AXIS_DRAD_EXTERNAL].stControl.bEnable := TRUE;

//B = A-E
fEncoderPosition := astAxes[AXIS_DRAD].stStatus.fActPosition - astAxes[AXIS_DRAD_INTERNAL].stStatus.fActPosition;
EncoderPosition:= LREAL_TO_DINT(fEncoderPosition * fScaler);

astAxes[AXIS_DRAD_EXTERNAL].stDescription.sAxisName := 'DRAD_EXTERNAL';

END_PROGRAM

// ---- POUs/Application_Specific/Axes/Virtuals/Drad_Internal.TcPOU
PROGRAM Drad_Internal
VAR
    fEncoderPosition : LREAL;
    EncoderPosition AT %Q* : DINT; //Encoder value for NC
    fScaler : LREAL := 100000;
END_VAR

GVL.astAxes[AXIS_DRAD_INTERNAL].stInputs.bLimitBwd := TRUE;
GVL.astAxes[AXIS_DRAD_INTERNAL].stInputs.bLimitFwd := TRUE;
GVL.astAxes[AXIS_DRAD_INTERNAL].stControl.bEnable := TRUE;

//E = SQRT(C^2 + F^2)


//calculate setpoint generator inputs
fEncoderPosition := SQRT(EXPT(astAxes[AXIS_DTANK_LENGTH].stStatus.fActPosition,2) + EXPT(astAxes[AXIS_DOFF_ANGLED].stStatus.fActPosition,2));
   
EncoderPosition:= LREAL_TO_DINT(fEncoderPosition * fScaler);

astAxes[AXIS_DRAD_INTERNAL].stDescription.sAxisName := 'DRAD_INTERNAL';

END_PROGRAM

// ---- POUs/Application_Specific/Axes/Virtuals/Doff_Angled.TcPOU
PROGRAM Doff_Angled
VAR
END_VAR

GVL.astAxes[AXIS_DOFF_ANGLED].stInputs.bLimitBwd := TRUE;
GVL.astAxes[AXIS_DOFF_ANGLED].stInputs.bLimitFwd := TRUE;
GVL.astAxes[AXIS_DOFF_ANGLED].stControl.bEnable := TRUE;

astAxes[AXIS_DOFF_ANGLED].stDescription.sAxisName := 'DOFF_ANGLED';

END_PROGRAM

// ---- POUs/Application_Specific/Axes/Virtuals/Doff_Parallel.TcPOU
PROGRAM Doff_Parallel
VAR
END_VAR

GVL.astAxes[AXIS_DOFF_PARALLEL].stInputs.bLimitBwd := TRUE;
GVL.astAxes[AXIS_DOFF_PARALLEL].stInputs.bLimitFwd := TRUE;
GVL.astAxes[AXIS_DOFF_PARALLEL].stControl.bEnable := TRUE;

astAxes[AXIS_DOFF_PARALLEL].stDescription.sAxisName := 'DOFF_PARALLEL';

END_PROGRAM

// ---- POUs/Application_Specific/Axes/Virtuals/Dtank_Internal_Offset_Angle.TcPOU
PROGRAM Dtank_Internal_Offset_Angle
VAR
    fEncoderPosition : LREAL;
    EncoderPosition AT %Q* : DINT; //Encoder value for NC
    fScaler : LREAL := 100000;
END_VAR

GVL.astAxes[AXIS_DTANK_INTERNAL_OFFSET_ANGLE].stInputs.bLimitBwd := TRUE;
GVL.astAxes[AXIS_DTANK_INTERNAL_OFFSET_ANGLE].stInputs.bLimitFwd := TRUE;
GVL.astAxes[AXIS_DTANK_INTERNAL_OFFSET_ANGLE].stControl.bEnable := TRUE;

//gamma = atan(F/C)

IF(astAxes[AXIS_DTANK_LENGTH].stStatus.fActPosition = 0) THEN
    fEncoderPosition:=0;
ELSE
    fEncoderPosition := RAD_TO_DEG(ATAN(astAxes[AXIS_DOFF_ANGLED].stStatus.fActPosition / astAxes[AXIS_DTANK_LENGTH].stStatus.fActPosition));
END_IF






   
EncoderPosition:= LREAL_TO_DINT(fEncoderPosition * fScaler);

astAxes[AXIS_DTANK_INTERNAL_OFFSET_ANGLE].stDescription.sAxisName := 'DRAD_INT_OFF';

END_PROGRAM

// ---- POUs/Application_Specific/Axes/Virtuals/Dtank_Length.TcPOU
PROGRAM Dtank_Length
VAR

END_VAR

GVL.astAxes[AXIS_DTANK_LENGTH].stInputs.bLimitBwd := TRUE;
GVL.astAxes[AXIS_DTANK_LENGTH].stInputs.bLimitFwd := TRUE;
GVL.astAxes[AXIS_DTANK_LENGTH].stControl.bEnable := TRUE;




IF _TaskInfo[fbGetCurTaskIndex.index].FirstCycle THEN
    //Initial default values:

END_IF


astAxes[AXIS_DTANK_LENGTH].stDescription.sAxisName := 'DTANK_LENGTH';

END_PROGRAM

// ---- POUs/Application_Specific/Axes/Virtuals/Dtank_Pivot_To_Window.TcPOU
PROGRAM Dtank_Pivot_To_Window
VAR

END_VAR

GVL.astAxes[AXIS_DTANK_PIVOT_TO_WINDOW].stInputs.bLimitBwd := TRUE;
GVL.astAxes[AXIS_DTANK_PIVOT_TO_WINDOW].stInputs.bLimitFwd := TRUE;
GVL.astAxes[AXIS_DTANK_PIVOT_TO_WINDOW].stControl.bEnable := TRUE;



IF _TaskInfo[fbGetCurTaskIndex.index].FirstCycle THEN
    //Initial default values:
END_IF

astAxes[AXIS_DTANK_PIVOT_TO_WINDOW].stDescription.sAxisName := 'PIVOT_TO_WINDOW';

END_PROGRAM

// ---- POUs/Application_Specific/Axes/Virtuals/Delta.TcPOU
PROGRAM Delta
VAR
END_VAR

GVL.astAxes[AXIS_DELTA].stInputs.bLimitBwd := TRUE;
GVL.astAxes[AXIS_DELTA].stInputs.bLimitFwd := TRUE;
GVL.astAxes[AXIS_DELTA].stControl.bEnable := TRUE;

astAxes[AXIS_DELTA].stDescription.sAxisName := 'DELTA';

END_PROGRAM

// ---- POUs/Application_Specific/Axes/Virtuals/Tau.TcPOU
PROGRAM Tau
VAR
    fEncoderPosition_tau : LREAL;
    EncoderPosition_tau AT %Q* : DINT; //Encoder value for NC
    fEncoderPosition_delta : LREAL;
    EncoderPosition_delta AT %Q* : DINT; //Encoder value for NC
    
    fScaler : LREAL := 100000;
    
    comp1 : LREAL; //holder
    comp2 : LREAL; //holder
END_VAR

GVL.astAxes[AXIS_TAU].stInputs.bLimitBwd := TRUE;
GVL.astAxes[AXIS_TAU].stInputs.bLimitFwd := TRUE;
GVL.astAxes[AXIS_TAU].stControl.bEnable := TRUE;


//C-D
comp1:= astAxes[AXIS_DTANK_LENGTH].stStatus.fActPosition - astAxes[AXIS_DTANK_PIVOT_TO_WINDOW].stStatus.fActPosition;

//F+G
comp2:= astAxes[AXIS_DOFF_ANGLED].stStatus.fActPosition + astAxes[AXIS_DOFF_PARALLEL].stStatus.fActPosition;

fEncoderPosition_tau := SQRT(EXPT(comp1,2)+EXPT(comp2,2));

IF comp1=0 THEN
    fEncoderPosition_delta := 0;
ELSE
    fEncoderPosition_delta := RAD_TO_DEG(ATAN(comp2/comp1));
END_IF


EncoderPosition_tau:= LREAL_TO_DINT(fEncoderPosition_tau * fScaler);
EncoderPosition_delta:= LREAL_TO_DINT(fEncoderPosition_delta * fScaler);

astAxes[AXIS_TAU].stDescription.sAxisName := 'TAU';

END_PROGRAM

// ---- POUs/Application_Specific/Axes/Virtuals/Drad.TcPOU
PROGRAM Drad
VAR
        //Requires feedback
    fEncoderPosition_DetectorArcRadius : LREAL;
    EncoderPosition_DetectorArcRadius AT %Q* : DINT;
    fEncoderPosition_MeasurementAngle : LREAL;
    EncoderPosition_MeasurementAngle AT %Q* : DINT;
    
    fScaler : LREAL := 100000;
    
    
    yPosition : LREAL;
    zPosition : LREAL;
    
    yPixelFromPivot : LREAL;
    zPixelFromPivot : LREAL;
    
END_VAR

GVL.astAxes[AXIS_DRAD].stInputs.bLimitBwd := TRUE;
GVL.astAxes[AXIS_DRAD].stInputs.bLimitFwd := TRUE;
GVL.astAxes[AXIS_DRAD].stControl.bEnable := TRUE;


yPixelFromPivot := -SIN(DEG_TO_RAD((astAxes[AXIS_DELTA].stStatus.fActPosition - astAxes[AXIS_MEASUREMENT_ANGLE].stStatus.fActPosition)))*astAxes[AXIS_TAU].stStatus.fActPosition;
zPixelFromPivot := COS(DEG_TO_RAD((astAxes[AXIS_DELTA].stStatus.fActPosition - astAxes[AXIS_MEASUREMENT_ANGLE].stStatus.fActPosition)))*astAxes[AXIS_TAU].stStatus.fActPosition;

yPosition := astAxes[AXIS_COMBINED_VERTICAL_VIRTUAL].stStatus.fActPosition + yPixelFromPivot;
zPosition := astAxes[AXIS_HORIZONTAL_VIRTUAL].stStatus.fActPosition + zPixelFromPivot; 

fEncoderPosition_DetectorArcRadius := SQRT(EXPT(yPosition,2)+EXPT(zPosition,2));
EncoderPosition_DetectorArcRadius := LREAL_TO_DINT(fEncoderPosition_DetectorArcRadius*fScaler);

IF zPosition = 0 THEN
    fEncoderPosition_MeasurementAngle := 0;
ELSE
    fEncoderPosition_MeasurementAngle := RAD_TO_DEG(ATAN(yPosition/zPosition));
END_IF


EncoderPosition_MeasurementAngle := LREAL_TO_DINT(fEncoderPosition_MeasurementAngle*fScaler);

IF _TaskInfo[fbGetCurTaskIndex.index].FirstCycle THEN
    //Initial default values:

END_IF

astAxes[AXIS_DRAD].stDescription.sAxisName := 'DRAD';

END_PROGRAM

// ---- POUs/Application_Specific/Axes/Virtuals/Measurement_Angle.TcPOU
PROGRAM Measurement_Angle
VAR
    //Feedback calculated in Detector Arc Radius prog
END_VAR

GVL.astAxes[AXIS_MEASUREMENT_ANGLE].stInputs.bLimitBwd := TRUE;
GVL.astAxes[AXIS_MEASUREMENT_ANGLE].stInputs.bLimitFwd := TRUE;
//GVL.astAxes[AXIS_MEASUREMENT_ANGLE].stControl.bEnable := TRUE;
astAxes[AXIS_MEASUREMENT_ANGLE].stDescription.sAxisName := 'MEASUREMENT_ANGLE';

END_PROGRAM

// ---- POUs/Application_Specific/Axes/Sample and Calibration/Rotation_Calibration.TcPOU
PROGRAM Rotation_Calibration
VAR
END_VAR

astAxes[AXIS_ROTATION_CALIBRATION].stControl.bEnable := TRUE;
astAxes[AXIS_ROTATION_CALIBRATION].stInputs.bLimitBwd := astAxes[AXIS_ROTATION].stInputs.bLimitBwd;
astAxes[AXIS_ROTATION_CALIBRATION].stInputs.bLimitFwd := astAxes[AXIS_ROTATION].stInputs.bLimitFwd;

astAxes[AXIS_ROTATION_CALIBRATION].stDescription.sAxisName := 'CALIB_ROT';

END_PROGRAM

// ---- POUs/Application_Specific/Axes/Sample and Calibration/Rotation_Sample.TcPOU
PROGRAM Rotation_Sample
VAR
END_VAR

astAxes[AXIS_ROTATION_SAMPLE].stControl.bEnable := TRUE;
astAxes[AXIS_ROTATION_SAMPLE].stInputs.bLimitBwd := astAxes[AXIS_ROTATION].stInputs.bLimitBwd;
astAxes[AXIS_ROTATION_SAMPLE].stInputs.bLimitFwd := astAxes[AXIS_ROTATION].stInputs.bLimitFwd;

astAxes[AXIS_ROTATION_SAMPLE].stDescription.sAxisName := 'SAMPLE_ROT';

END_PROGRAM

// ---- POUs/Application_Specific/Axes/Sample and Calibration/Horizontal_Calibration.TcPOU
PROGRAM Horizontal_Calibration
VAR
END_VAR

astAxes[AXIS_HORIZONTAL_CALIBRATION].stControl.bEnable := TRUE;
astAxes[AXIS_HORIZONTAL_CALIBRATION].stInputs.bLimitBwd := astAxes[AXIS_HORIZONTAL_TRANSLATION].stInputs.bLimitBwd;
astAxes[AXIS_HORIZONTAL_CALIBRATION].stInputs.bLimitFwd := astAxes[AXIS_HORIZONTAL_TRANSLATION].stInputs.bLimitFwd;

astAxes[AXIS_HORIZONTAL_CALIBRATION].stDescription.sAxisName := 'CALIB_HORIZ';

END_PROGRAM

// ---- POUs/Application_Specific/Axes/Sample and Calibration/Horizontal_Sample.TcPOU
PROGRAM Horizontal_Sample
VAR
END_VAR

astAxes[AXIS_HORIZONTAL_SAMPLE].stControl.bEnable := TRUE;
astAxes[AXIS_HORIZONTAL_SAMPLE].stInputs.bLimitBwd := astAxes[AXIS_HORIZONTAL_TRANSLATION].stInputs.bLimitBwd;
astAxes[AXIS_HORIZONTAL_SAMPLE].stInputs.bLimitFwd := astAxes[AXIS_HORIZONTAL_TRANSLATION].stInputs.bLimitFwd;

astAxes[AXIS_HORIZONTAL_SAMPLE].stDescription.sAxisName := 'SAMPLE_HORIZ';

END_PROGRAM

// ---- POUs/Application_Specific/Axes/Sample and Calibration/Combined_Vertical_Calibration.TcPOU
PROGRAM Combined_Vertical_Calibration
VAR
END_VAR

astAxes[AXIS_COMBINED_VERTICAL_CALIBRATION].stControl.bEnable := TRUE;
astAxes[AXIS_COMBINED_VERTICAL_CALIBRATION].stInputs.bLimitBwd := astAxes[AXIS_COMBINED_VERTICAL].stInputs.bLimitBwd;
astAxes[AXIS_COMBINED_VERTICAL_CALIBRATION].stInputs.bLimitFwd := astAxes[AXIS_COMBINED_VERTICAL].stInputs.bLimitFwd;

astAxes[AXIS_COMBINED_VERTICAL_CALIBRATION].stDescription.sAxisName := 'CALIB_Y';

END_PROGRAM

// ---- POUs/Application_Specific/Axes/Sample and Calibration/Combined_Vertical_Sample.TcPOU
PROGRAM Combined_Vertical_Sample
VAR
END_VAR

astAxes[AXIS_COMBINED_VERTICAL_SAMPLE].stControl.bEnable := TRUE;
astAxes[AXIS_COMBINED_VERTICAL_SAMPLE].stInputs.bLimitBwd := astAxes[AXIS_COMBINED_VERTICAL].stInputs.bLimitBwd;
astAxes[AXIS_COMBINED_VERTICAL_SAMPLE].stInputs.bLimitFwd := astAxes[AXIS_COMBINED_VERTICAL].stInputs.bLimitFwd;

astAxes[AXIS_COMBINED_VERTICAL_SAMPLE].stDescription.sAxisName := 'SAMPLE_Y';

END_PROGRAM

// ---- POUs/Application_Specific/Axes/Sample and Calibration/Measurement_Angle_Offset.TcPOU
PROGRAM Measurement_Angle_Offset
VAR
END_VAR

astAxes[AXIS_MEASUREMENT_ANGLE_OFFSET].stInputs.bLimitBwd := TRUE;
astAxes[AXIS_MEASUREMENT_ANGLE_OFFSET].stInputs.bLimitFwd := TRUE;
astAxes[AXIS_MEASUREMENT_ANGLE_OFFSET].stControl.bEnable:= TRUE;

astAxes[AXIS_MEASUREMENT_ANGLE_OFFSET].stDescription.sAxisName := 'OFFSET_MEAS_ANGLE';

END_PROGRAM

// ---- POUs/Application_Specific/Axes/Real axis follows/Rotation_Virtual.TcPOU
PROGRAM Rotation_Virtual
VAR
    fEncoderPosition : LREAL;
    EncoderPosition AT %Q* : DINT; //Encoder value for NC
    fScaler : LREAL := 100000;
END_VAR

GVL.astAxes[AXIS_ROTATION_VIRTUAL].stInputs.bLimitBwd := TRUE;
GVL.astAxes[AXIS_ROTATION_VIRTUAL].stInputs.bLimitFwd := TRUE;
GVL.astAxes[AXIS_ROTATION_VIRTUAL].stControl.bEnable := TRUE;




//calculate setpoint generator inputs
fEncoderPosition := 
    GVL_INTER.TARGET_MEASUREMENT_ANGLE +
    astAxes[AXIS_DTANK_INTERNAL_OFFSET_ANGLE].Axis.NcToPlc.ActPos;
   
EncoderPosition:= LREAL_TO_DINT(fEncoderPosition * fScaler);

//astAxes[].stStatus.fActPosition
astAxes[AXIS_ROTATION_VIRTUAL].stDescription.sAxisName := 'ROT_VIRT';

END_PROGRAM

// ---- POUs/Application_Specific/Axes/Real axis follows/Combined_Vertical_Virtual.TcPOU
PROGRAM Combined_Vertical_Virtual
VAR
    fEncoderPosition : LREAL;
    EncoderPosition AT %Q* : DINT; //Encoder value for NC
    fScaler : LREAL := 100000;
END_VAR

GVL.astAxes[AXIS_COMBINED_VERTICAL_VIRTUAL].stInputs.bLimitBwd := TRUE;
GVL.astAxes[AXIS_COMBINED_VERTICAL_VIRTUAL].stInputs.bLimitFwd := TRUE;
GVL.astAxes[AXIS_COMBINED_VERTICAL_VIRTUAL].stControl.bEnable := TRUE;




//calculate setpoint generator inputs
fEncoderPosition := 
    astAxes[AXIS_DRAD_EXTERNAL].Axis.NcToPlc.ActPos * SIN(DEG_TO_RAD(GVL_INTER.TARGET_MEASUREMENT_ANGLE)) +
    astAxes[AXIS_DTANK_PIVOT_TO_WINDOW].Axis.NcToPlc.SetPos * SIN(DEG_TO_RAD(GVL_INTER.TARGET_MEASUREMENT_ANGLE + astAxes[AXIS_DTANK_INTERNAL_OFFSET_ANGLE].Axis.NcToPlc.ActPos)) +
    astAxes[AXIS_DOFF_PARALLEL].Axis.NcToPlc.SetPos * COS(DEG_TO_RAD(GVL_INTER.TARGET_MEASUREMENT_ANGLE + astAxes[AXIS_DTANK_INTERNAL_OFFSET_ANGLE].Axis.NcToPlc.ActPos)); 
    
EncoderPosition:= LREAL_TO_DINT(fEncoderPosition * fScaler);    

astAxes[AXIS_COMBINED_VERTICAL_VIRTUAL].stDescription.sAxisName := 'COMBINED_Y_VIRT';

END_PROGRAM

// ---- POUs/Application_Specific/Axes/Real axis follows/Horizontal_Virtual.TcPOU
PROGRAM Horizontal_Virtual
VAR
    fEncoderPosition : LREAL;
    EncoderPosition AT %Q* : DINT; //Encoder value for NC
    fScaler : LREAL := 100000;
END_VAR

GVL.astAxes[AXIS_HORIZONTAL_VIRTUAL].stInputs.bLimitBwd := TRUE;
GVL.astAxes[AXIS_HORIZONTAL_VIRTUAL].stInputs.bLimitFwd := TRUE;
GVL.astAxes[AXIS_HORIZONTAL_VIRTUAL].stControl.bEnable := TRUE;




//calculate setpoint generator inputs
fEncoderPosition := 
    astAxes[AXIS_DRAD_EXTERNAL].Axis.NcToPlc.ActPos * COS(DEG_TO_RAD(GVL_INTER.TARGET_MEASUREMENT_ANGLE)) +
    astAxes[AXIS_DTANK_PIVOT_TO_WINDOW].Axis.NcToPlc.SetPos * COS(DEG_TO_RAD(GVL_INTER.TARGET_MEASUREMENT_ANGLE + astAxes[AXIS_DTANK_INTERNAL_OFFSET_ANGLE].Axis.NcToPlc.ActPos)) -
    astAxes[AXIS_DOFF_PARALLEL].Axis.NcToPlc.SetPos * SIN(DEG_TO_RAD(GVL_INTER.TARGET_MEASUREMENT_ANGLE + astAxes[AXIS_DTANK_INTERNAL_OFFSET_ANGLE].Axis.NcToPlc.ActPos)); 
    
EncoderPosition:= LREAL_TO_DINT(fEncoderPosition * fScaler);    

astAxes[AXIS_HORIZONTAL_VIRTUAL].stDescription.sAxisName := 'HORIZ_VIRT';

END_PROGRAM

// ---- POUs/Application_Specific/Applications/INTER_LOGIC.TcPOU
PROGRAM INTER_LOGIC
VAR
    checkRotationDrive : MC_ReadStatus;
    IDs_RealAxes : ARRAY[1..ARRAYSIZE_REAL] OF UINT:= 
        [AXIS_HORIZONTAL_TRANSLATION,AXIS_COMBINED_VERTICAL,AXIS_ROTATION];
    vertTon : TON;
    
    LOCALMODE_SPEED_OVERRIDE : LREAL := 20; //Local mode override of base 20%
    LOCALMODE_SPEED_OVERRIDE_MODIFIER : LREAL := 1; //Proportional modifier to local mode speed
    
    //arraysSetup : BOOL := FALSE;
    driveStartupDelay : TON;

    
    safetyFTrig : F_TRIG;
    safetyResetTON : TON;
    safetyResetLatch : BOOL :=FALSE;
    safetyResetDone: BOOL;
    driveResetDone : BOOL;
    bRotationValid : BOOL:= FALSE;
    setPosRotation : MC_SetPosition;
    
    
    CombinedVerticalSetupComplete : BOOL := FALSE;
    AllowedVerticalLag : LREAL := 0.2;  //How much offset is allowed between two vertical axes when synced
    VerticalAxesCalibrated : BOOL := FALSE;
    VerticalAxesSpgEnabled : BOOL := FALSE;
    
    verticalZ1SpgEnable : MC_ExtSetPointGenEnable;
    verticalZ1SpgDisable : MC_ExtSetPointGenDisable;
    verticalZ2SpgEnable : MC_ExtSetPointGenEnable;
    verticalZ2SpgDisable : MC_ExtSetPointGenDisable;
    
    
    combinedVerticalSetPos : MC_SetPosition();
    
    eStateVertical : eState_Vertical := eState_Vertical.init;
    fVerticalSimulatedDeviation : LREAL;
    fVerticalSimulatedDeviationAllowed : LREAL := 0.1;
    confirmSpgTimeout : TON;
    fY1_To_Simulated_Deviation : LREAL;
    fY2_To_Simulated_Deviation : LREAL;
    y1Compensating : BOOL;
    y2Compensating : BOOL;
    fY1_To_Simulated_Deviation_Latched : LREAL;
    fY2_To_Simulated_Deviation_Latched : LREAL;
    y1CompensatingCycle : LREAL;
    y2CompensatingCycle : LREAL;
    CYCLES_TO_COMPENSATE : LREAL := 500;
    y1NotFinished : BOOL;
    y2NotFinished : BOOL;
    
    tempZ1Power : MC_Power;
    tempZ2Power : MC_Power;
    
    fZ1SetPos : LREAL;
    fZ1SetVelo : LREAL;
    fZ2SetPos : LREAL;
    fZ2SetVelo : LREAL;
    fZ1SetDir : DINT;
    fZ2SetDir : DINT;
    combinedVerticalDirection : DINT;
    

    imHere: INT;
    
    
    
    //////////////////////////////////////////////////
    
    //SETPOINT GENERATORS FOR KINEMATICS
    axisSpg_Vertical : ST_AxisSpg:= (axisID:= AXIS_COMBINED_VERTICAL);
    axisSpg_Horizontal : ST_AxisSpg:= (axisID:= AXIS_HORIZONTAL_TRANSLATION);
    axisSpg_Rot : ST_AxisSpg:= (axisID:= AXIS_ROTATION);
    enableSPGs : BOOL;
    disableSPGs : BOOL; 
        
    /////////////////////////
    eStateInter : eState_INTER := eState_INTER.init;
    checkFirstCycle : BOOL;
    posDevHorizontal : LREAL;
    posDevVertical : LREAL;
    posDevRot : LREAL;
    bRealDevValid : BOOL;
    bDefaultDevValid : BOOL;
    bRecoveryDevValid : BOOL;
    /////////////////////////
    
    bKinematicsOperational : BOOL;
    bVirtualsMoving : BOOL;
    writeDefault : FB_WritePersistentData;
    
    startupDelayTON : TON;
    timeoutDelay : TON;
    stateDelayTimer : TON;
    retryCounter : INT := 0;
    
    i : INT :=0; //iterator for FOR loops
    bVertCorrectionInProgress : BOOL;
    vertDelay : TON;
END_VAR

VAR CONSTANT
    DEVIATION_THRESHOLD : LREAL := 0.05;
    ARRAYSIZE_REAL : INT := 3;
    ARRAYSIZE_VIRTUALCAL : INT :=3;
    ARRAYSIZE_VIRTUAL : INT:= 10;
    ARRAYSIZE_ALLVIRTUALS : INT:= 13;
    VERTICAL_SPEED_LIMIT :LREAL := 4;
    HORIZONTAL_SPEED_LIMIT:LREAL:= 4;
    ROTATION_SPEED_LIMIT :LREAL:= 0.1;
END_VAR

VAR PERSISTENT   
    aVirtualAxisDefaults : ARRAY [1..ARRAYSIZE_ALLVIRTUALS] OF ST_DefaultVals:=
    [(axisID:=AXIS_DRAD, defaultPosition:=3000),
     (axisID:=AXIS_DTANK_LENGTH, defaultPosition:=2289.15),
    (axisID:=AXIS_DTANK_PIVOT_TO_WINDOW, defaultPosition:=1648.66),
    (axisID:=AXIS_MEASUREMENT_ANGLE, defaultPosition:=0),
    (axisID:=AXIS_DOFF_ANGLED, defaultPosition:=0),
    (axisID:=AXIS_DOFF_PARALLEL, defaultPosition:=0),
    (axisID:=AXIS_HORIZONTAL_CALIBRATION, defaultPosition:=0),
    (axisID:=AXIS_HORIZONTAL_SAMPLE, defaultPosition:=0),
    (axisID:=AXIS_COMBINED_VERTICAL_CALIBRATION, defaultPosition:=0),
    (axisID:=AXIS_COMBINED_VERTICAL_SAMPLE, defaultPosition:=0),
    (axisID:=AXIS_ROTATION_CALIBRATION, defaultPosition:=0),
    (axisID:=AXIS_ROTATION_SAMPLE, defaultPosition:=0),
    (axisID:=AXIS_MEASUREMENT_ANGLE_OFFSET, defaultPosition:=0)]
;
END_VAR

actSafeSpeedSwitching();
IF GVL_INTER.ENABLE_ALL_AXES THEN
    EnableAxes();
END_IF

IF GVL_INTER.DISABLE_ALL_AXES THEN
    DisableAxes();
END_IF

safetyFTrig(CLK:= GVL_Safety.ResetPossibleAndPressed);
IF safetyFTrig.Q THEN
    safetyResetLatch := TRUE;
    safetyResetDone:= FALSE;
    driveResetDone:= FALSE;
END_IF

safetyResetTON(IN:= safetyResetLatch, PT:=T#1S);
driveStartupDelay(IN:=safetyResetLatch,  PT:=T#2S);

IF safetyResetTON.Q THEN
    safetyResetDone := TRUE;
    GVL_INTER.RESET_ALL := TRUE;
END_IF

IF driveStartupDelay.Q THEN
    driveResetDone := TRUE;
END_IF

IF driveResetDone AND safetyResetDone THEN
    safetyResetLatch:= FALSE;
END_IF

IF GVL_INTER.RESET_ALL THEN
    ResetAll();
END_IF

GVL_INTER.NC_AXIS_ERROR := CheckNcErrors();
VerticalAxesCalibrated := CheckVerticalCalibration();
VerticalAxesSpgEnabled := CheckZSpgStatus();
GVL_INTER.LIMIT_HIT:= CheckRealLimits();

CombinedVerticalSetupComplete := FALSE;
IF GVL_INTER.RUN_COUPLED_VERTICAL AND driveResetDone THEN      
    //Enable linking
    IF astAxes[AXIS_VERTICAL_TRANSLATION_Y2].stStatus.bEnabled AND astAxes[AXIS_VERTICAL_TRANSLATION_Y1].stStatus.bEnabled THEN
        IF VerticalAxesCalibrated AND  VerticalAxesSpgEnabled AND NOT (astAxes[AXIS_VERTICAL_TRANSLATION_Y1].stStatus.bError OR astAxes[AXIS_VERTICAL_TRANSLATION_Y2].stStatus.bError)THEN
            astAxes[AXIS_COMBINED_VERTICAL].stControl.bEnable := TRUE;
        ELSE 
            astAxes[AXIS_COMBINED_VERTICAL].stControl.bEnable := FALSE;
		END_IF
	END_IF
    
    //Fwd limit linking
    astAxes[AXIS_COMBINED_VERTICAL].stInputs.bLimitFwd := (astAxes[AXIS_VERTICAL_TRANSLATION_Y2].stInputs.bLimitFwd AND astAxes[AXIS_VERTICAL_TRANSLATION_Y1].stInputs.bLimitFwd);
    astAxes[AXIS_COMBINED_VERTICAL].stInputs.bLimitBwd := (astAxes[AXIS_VERTICAL_TRANSLATION_Y2].stInputs.bLimitBwd AND astAxes[AXIS_VERTICAL_TRANSLATION_Y1].stInputs.bLimitBwd);
    
    IF NOT GVL_INTER.DECOUPLE_VERTICAL_AXES THEN
        astAxes[AXIS_VERTICAL_TRANSLATION_Y2].stInputs.bLimitFwd := TRUE;
        astAxes[AXIS_VERTICAL_TRANSLATION_Y2].stInputs.bLimitBwd := TRUE;
        astAxes[AXIS_VERTICAL_TRANSLATION_Y1].stInputs.bLimitFwd := TRUE;
        astAxes[AXIS_VERTICAL_TRANSLATION_Y1].stInputs.bLimitBwd := TRUE;
	END_IF
    
    fVerticalSimulatedDeviation := astAxes[AXIS_COMBINED_VERTICAL].stStatus.fActPosition - astAxes[AXIS_VERTICAL_TRANSLATION_Y1].stStatus.fActPosition;
    
    confirmSpgTimeout(PT:=T#1S);

    
    IF astAxes[AXIS_VERTICAL_TRANSLATION_Y1].stStatus.bError OR astAxes[AXIS_VERTICAL_TRANSLATION_Y2].stStatus.bError THEN
        eStateVertical:= eState_Vertical.init;
	END_IF
    
    actSyncVertStateMachine();
        
END_IF

combinedVerticalSetPos(Axis:= astAxes[AXIS_COMBINED_VERTICAL].Axis);
combinedVerticalSetPos.Execute:= FALSE;

IF(astAxes[AXIS_COMBINED_VERTICAL].Axis.NcToPlc.ActVelo>0) THEN
    combinedVerticalDirection := 1;
ELSIF (astAxes[AXIS_COMBINED_VERTICAL].Axis.NcToPlc.ActVelo<0) THEN
    combinedVerticalDirection := -1;
ELSE 
    combinedVerticalDirection := 0;
END_IF

actZSetpoints();
verticalZ1SpgEnable(Axis:=astAxes[AXIS_VERTICAL_TRANSLATION_Y1].Axis);
verticalZ1SpgEnable.Execute:= FALSE;
verticalZ1SpgDisable(Axis:=astAxes[AXIS_VERTICAL_TRANSLATION_Y1].Axis);
verticalZ1SpgDisable.Execute:= FALSE;
verticalZ2SpgEnable(Axis:=astAxes[AXIS_VERTICAL_TRANSLATION_Y2].Axis);
verticalZ2SpgEnable.Execute:= FALSE;
verticalZ2SpgDisable(Axis:=astAxes[AXIS_VERTICAL_TRANSLATION_Y2].Axis);
verticalZ2SpgDisable.Execute:= FALSE;

writeDefault(NETID:='', PORT:=852);
writeDefault.START:= FALSE;


